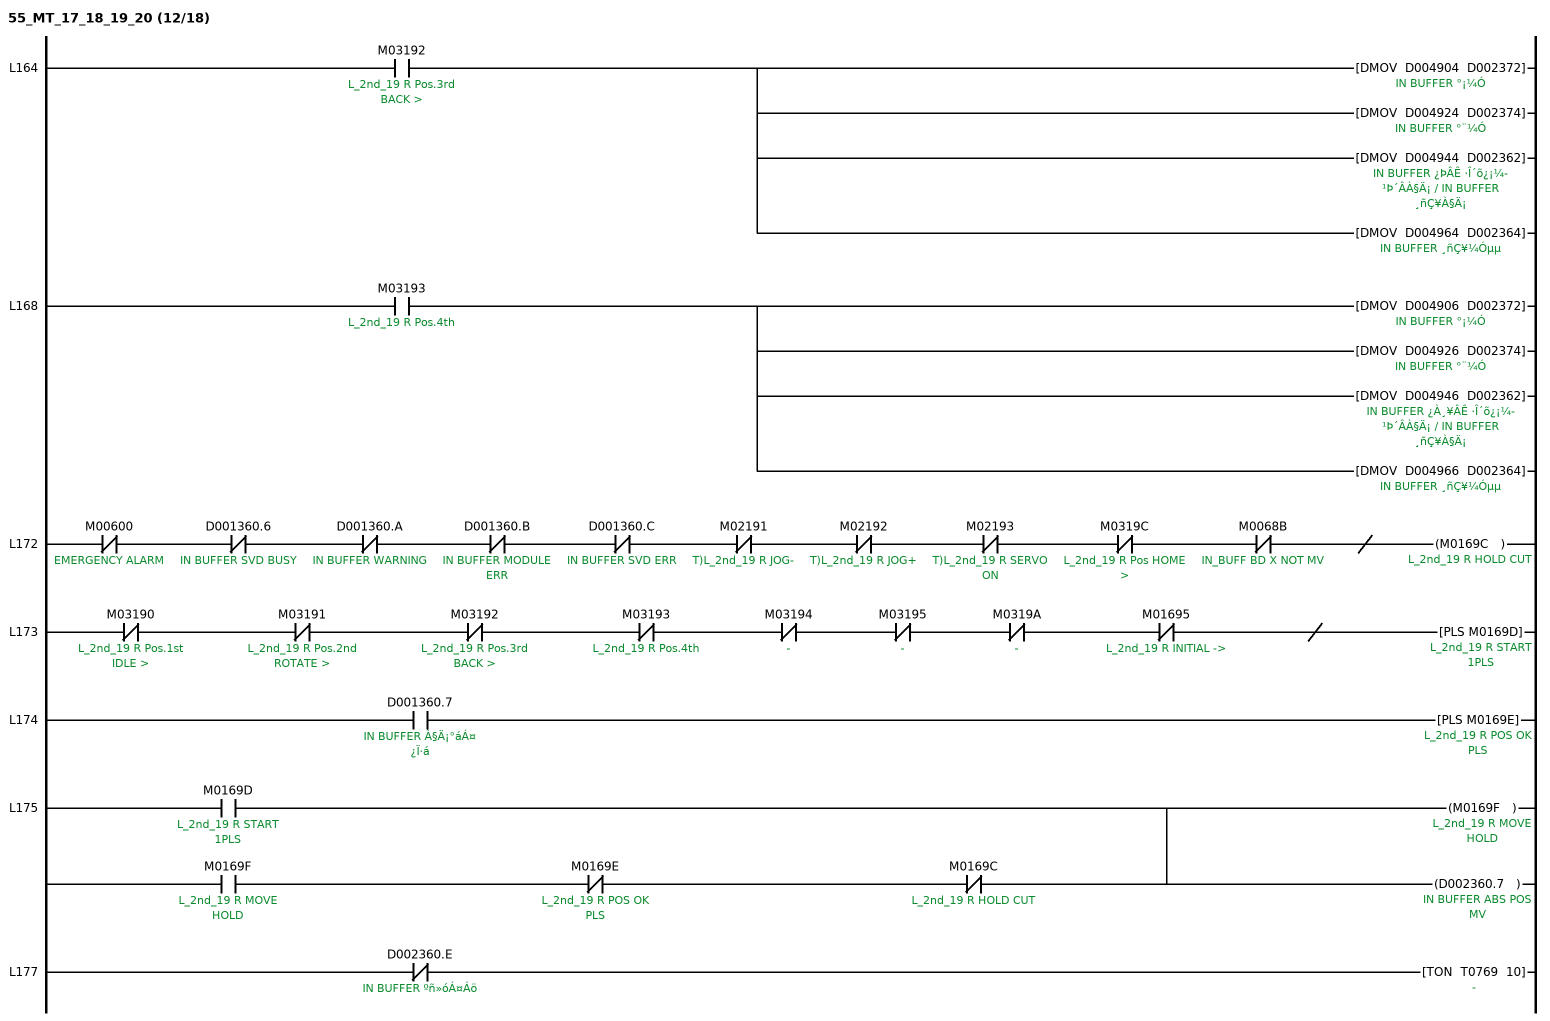
[picture p336: 55_MT_17_18_19_20 rungs L164-L177]
; L164
LOAD      M03192	// L_2nd_19 R Pos.3rd BACK >
DMOV      D004904 D002372	// IN BUFFER °¡¼Ó
DMOV      D004924 D002374	// IN BUFFER °¨¼Ó
DMOV      D004944 D002362	// IN BUFFER ¿ÞÂÊ ·Î´õ¿¡¼­ ¹Þ´ÂÀ§Ä¡ / IN BUFFER ¸ñÇ¥À§Ä¡
DMOV      D004964 D002364	// IN BUFFER ¸ñÇ¥¼Óµµ
; L168
LOAD      M03193	// L_2nd_19 R Pos.4th 
DMOV      D004906 D002372	// IN BUFFER °¡¼Ó
DMOV      D004926 D002374	// IN BUFFER °¨¼Ó
DMOV      D004946 D002362	// IN BUFFER ¿À¸¥ÂÊ ·Î´õ¿¡¼­ ¹Þ´ÂÀ§Ä¡ / IN BUFFER ¸ñÇ¥À§Ä¡
DMOV      D004966 D002364	// IN BUFFER ¸ñÇ¥¼Óµµ
; L172
LOAD NOT  M00600	// EMERGENCY ALARM
AND NOT   D001360.6	// IN BUFFER SVD BUSY
AND NOT   D001360.A	// IN BUFFER WARNING
AND NOT   D001360.B	// IN BUFFER MODULE ERR
AND NOT   D001360.C	// IN BUFFER SVD ERR
AND NOT   M02191	// T)L_2nd_19 R JOG-
AND NOT   M02192	// T)L_2nd_19 R JOG+
AND NOT   M02193	// T)L_2nd_19 R SERVO ON
AND NOT   M0319C	// L_2nd_19 R Pos HOME >
AND NOT   M0068B	// IN_BUFF BD X NOT MV
NOT
OUT       M0169C	// L_2nd_19 R HOLD CUT
; L173
LOAD NOT  M03190	// L_2nd_19 R Pos.1st IDLE >
AND NOT   M03191	// L_2nd_19 R Pos.2nd ROTATE >
AND NOT   M03192	// L_2nd_19 R Pos.3rd BACK >
AND NOT   M03193	// L_2nd_19 R Pos.4th 
AND NOT   M03194	// -
AND NOT   M03195	// -
AND NOT   M0319A	// -
AND NOT   M01695	// L_2nd_19 R INITIAL ->
NOT
OUTP      M0169D	// L_2nd_19 R START 1PLS
; L174
LOAD      D001360.7	// IN BUFFER À§Ä¡°áÁ¤ ¿Ï·á
OUTP      M0169E	// L_2nd_19 R POS OK PLS
; L175
LOAD      M0169D	// L_2nd_19 R START 1PLS
LOAD      M0169F	// L_2nd_19 R MOVE HOLD
AND NOT   M0169E	// L_2nd_19 R POS OK PLS
AND NOT   M0169C	// L_2nd_19 R HOLD CUT
OR LOAD
OUT       M0169F	// L_2nd_19 R MOVE HOLD
OUT       D002360.7	// IN BUFFER ABS POS MV
; L177
LOAD NOT  D002360.E	// IN BUFFER ºñ»óÁ¤Áö
TON       T0769 10	// -

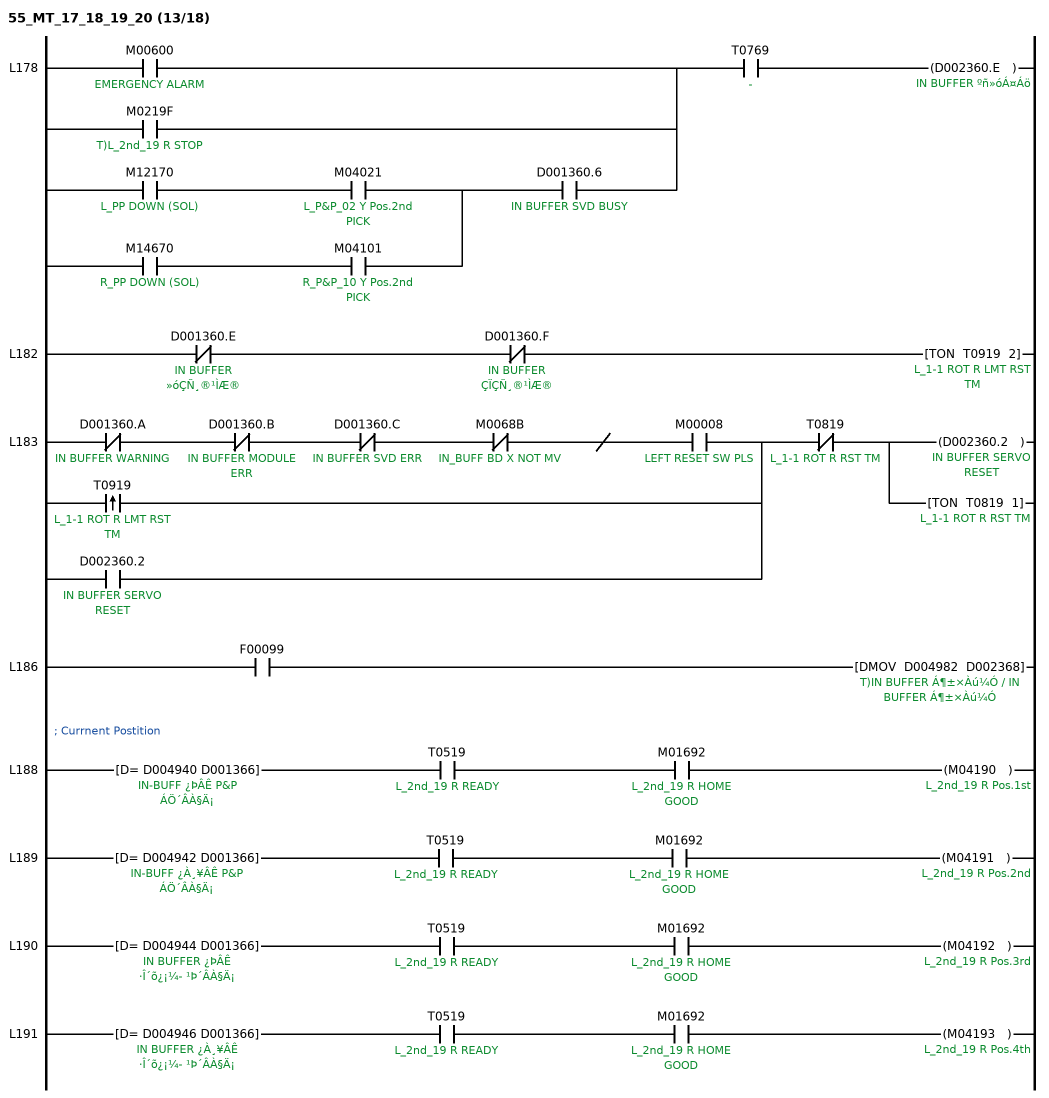
; L178
LOAD      M00600	// EMERGENCY ALARM
OR        M0219F	// T)L_2nd_19 R STOP
LOAD      M12170	// L_PP DOWN (SOL)
AND       M04021	// L_P&P_02 Y Pos.2nd PICK
LOAD      M14670	// R_PP DOWN (SOL)
AND       M04101	// R_P&P_10 Y Pos.2nd PICK
OR LOAD
AND       D001360.6	// IN BUFFER SVD BUSY
OR LOAD
AND       T0769	// -
OUT       D002360.E	// IN BUFFER ºñ»óÁ¤Áö
; L182
LOAD NOT  D001360.E	// IN BUFFER »óÇÑ¸®¹ÌÆ®
AND NOT   D001360.F	// IN BUFFER ÇÏÇÑ¸®¹ÌÆ®
TON       T0919 2	// L_1-1 ROT R LMT RST TM
; L183
LOAD NOT  D001360.A	// IN BUFFER WARNING
AND NOT   D001360.B	// IN BUFFER MODULE ERR
AND NOT   D001360.C	// IN BUFFER SVD ERR
AND NOT   M0068B	// IN_BUFF BD X NOT MV
NOT
AND       M00008	// LEFT RESET SW PLS
ORP       T0919	// L_1-1 ROT R LMT RST TM
OR        D002360.2	// IN BUFFER SERVO RESET
AND NOT   T0819	// L_1-1 ROT R RST TM
OUT       D002360.2	// IN BUFFER SERVO RESET
TON       T0819 1	// L_1-1 ROT R RST TM
; L186
LOAD      F00099
DMOV      D004982 D002368	// T)IN BUFFER Á¶±×Àú¼Ó / IN BUFFER Á¶±×Àú¼Ó
// Currnent Postition
; L188
LOADD=    D004940 D001366	// IN-BUFF ¿ÞÂÊ P&P ÁÖ´ÂÀ§Ä¡
AND       T0519	// L_2nd_19 R READY
AND       M01692	// L_2nd_19 R HOME GOOD
OUT       M04190	// L_2nd_19 R Pos.1st 
; L189
LOADD=    D004942 D001366	// IN-BUFF ¿À¸¥ÂÊ P&P ÁÖ´ÂÀ§Ä¡
AND       T0519	// L_2nd_19 R READY
AND       M01692	// L_2nd_19 R HOME GOOD
OUT       M04191	// L_2nd_19 R Pos.2nd
; L190
LOADD=    D004944 D001366	// IN BUFFER ¿ÞÂÊ ·Î´õ¿¡¼­ ¹Þ´ÂÀ§Ä¡
AND       T0519	// L_2nd_19 R READY
AND       M01692	// L_2nd_19 R HOME GOOD
OUT       M04192	// L_2nd_19 R Pos.3rd
; L191
LOADD=    D004946 D001366	// IN BUFFER ¿À¸¥ÂÊ ·Î´õ¿¡¼­ ¹Þ´ÂÀ§Ä¡
AND       T0519	// L_2nd_19 R READY
AND       M01692	// L_2nd_19 R HOME GOOD
OUT       M04193	// L_2nd_19 R Pos.4th 

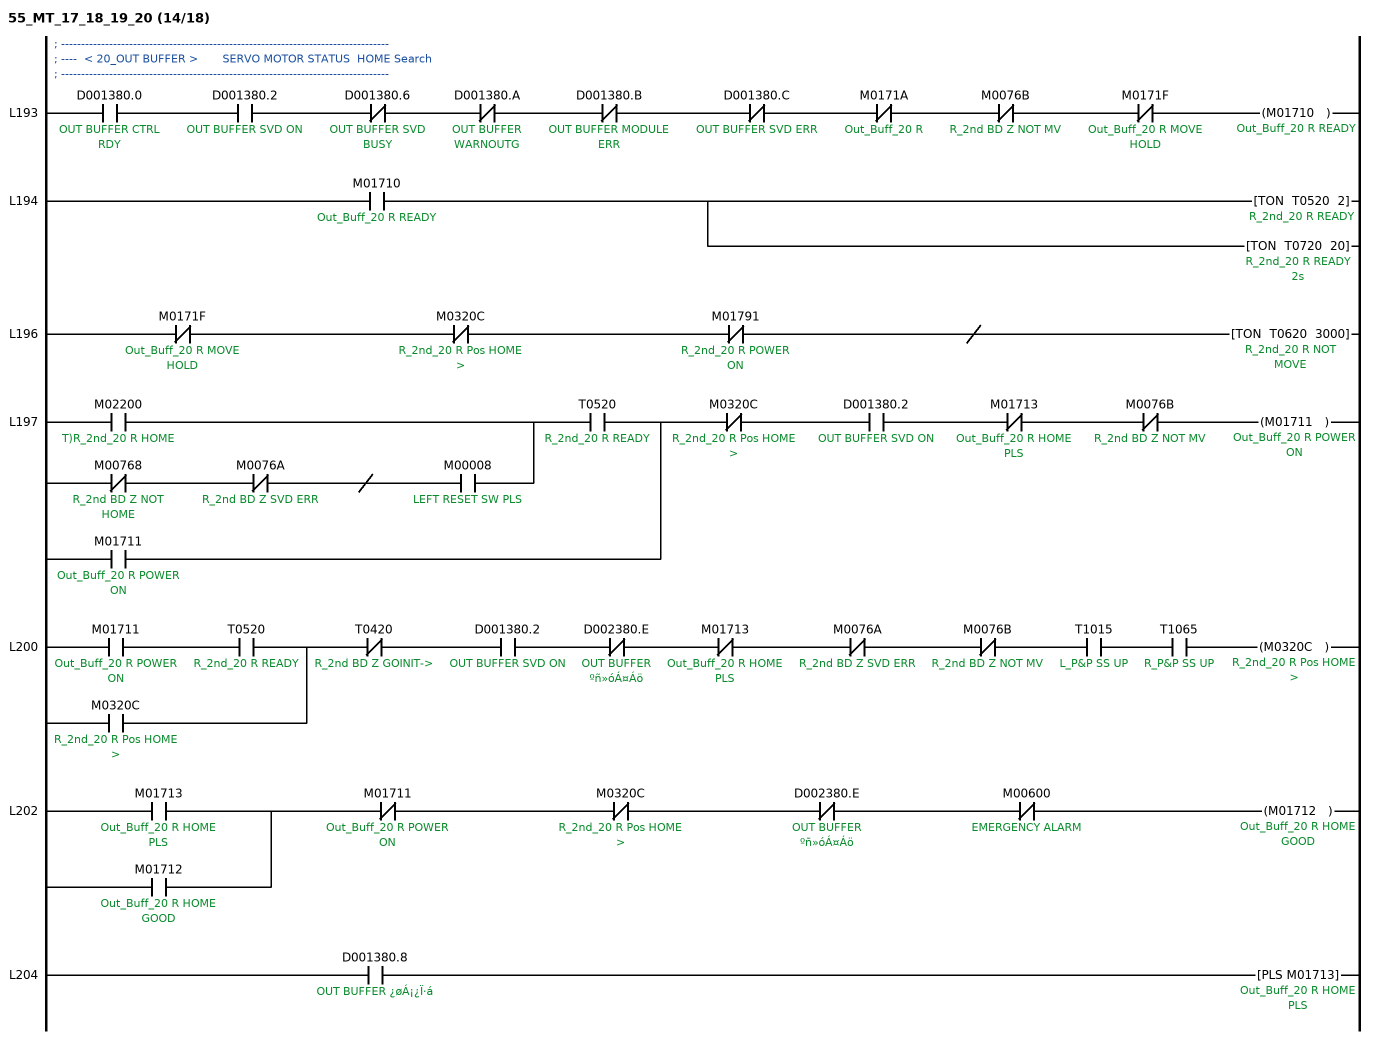
// ----------------------------------------------------------------------------------
// 
// ----  < 20_OUT BUFFER >       SERVO MOTOR STATUS  HOME Search
// 
// ----------------------------------------------------------------------------------
; L193
LOAD      D001380.0	// OUT BUFFER CTRL RDY
AND       D001380.2	// OUT BUFFER SVD ON
AND NOT   D001380.6	// OUT BUFFER SVD BUSY
AND NOT   D001380.A	// OUT BUFFER WARNOUTG
AND NOT   D001380.B	// OUT BUFFER MODULE ERR
AND NOT   D001380.C	// OUT BUFFER SVD ERR
AND NOT   M0171A	// Out_Buff_20 R
AND NOT   M0076B	// R_2nd BD Z NOT MV
AND NOT   M0171F	// Out_Buff_20 R MOVE HOLD
OUT       M01710	// Out_Buff_20 R READY
; L194
LOAD      M01710	// Out_Buff_20 R READY
TON       T0520 2	// R_2nd_20 R READY
TON       T0720 20	// R_2nd_20 R READY 2s
; L196
LOAD NOT  M0171F	// Out_Buff_20 R MOVE HOLD
AND NOT   M0320C	// R_2nd_20 R Pos HOME >
AND NOT   M01791	// R_2nd_20 R POWER ON
NOT
TON       T0620 3000	// R_2nd_20 R NOT MOVE
; L197
LOAD      M02200	// T)R_2nd_20 R HOME
LOAD NOT  M00768	// R_2nd BD Z NOT HOME
AND NOT   M0076A	// R_2nd BD Z SVD ERR
NOT
AND       M00008	// LEFT RESET SW PLS
OR LOAD
AND       T0520	// R_2nd_20 R READY
OR        M01711	// Out_Buff_20 R POWER ON
AND NOT   M0320C	// R_2nd_20 R Pos HOME >
AND       D001380.2	// OUT BUFFER SVD ON
AND NOT   M01713	// Out_Buff_20 R HOME PLS
AND NOT   M0076B	// R_2nd BD Z NOT MV
OUT       M01711	// Out_Buff_20 R POWER ON
; L200
LOAD      M01711	// Out_Buff_20 R POWER ON
AND       T0520	// R_2nd_20 R READY
OR        M0320C	// R_2nd_20 R Pos HOME >
AND NOT   T0420	// R_2nd BD Z GOINIT->
AND       D001380.2	// OUT BUFFER SVD ON
AND NOT   D002380.E	// OUT BUFFER ºñ»óÁ¤Áö
AND NOT   M01713	// Out_Buff_20 R HOME PLS
AND NOT   M0076A	// R_2nd BD Z SVD ERR
AND NOT   M0076B	// R_2nd BD Z NOT MV
AND       T1015	// L_P&P SS UP
AND       T1065	// R_P&P SS UP
OUT       M0320C	// R_2nd_20 R Pos HOME >
; L202
LOAD      M01713	// Out_Buff_20 R HOME PLS
OR        M01712	// Out_Buff_20 R HOME GOOD
AND NOT   M01711	// Out_Buff_20 R POWER ON
AND NOT   M0320C	// R_2nd_20 R Pos HOME >
AND NOT   D002380.E	// OUT BUFFER ºñ»óÁ¤Áö
AND NOT   M00600	// EMERGENCY ALARM
OUT       M01712	// Out_Buff_20 R HOME GOOD
; L204
LOAD      D001380.8	// OUT BUFFER ¿øÁ¡¿Ï·á
OUTP      M01713	// Out_Buff_20 R HOME PLS

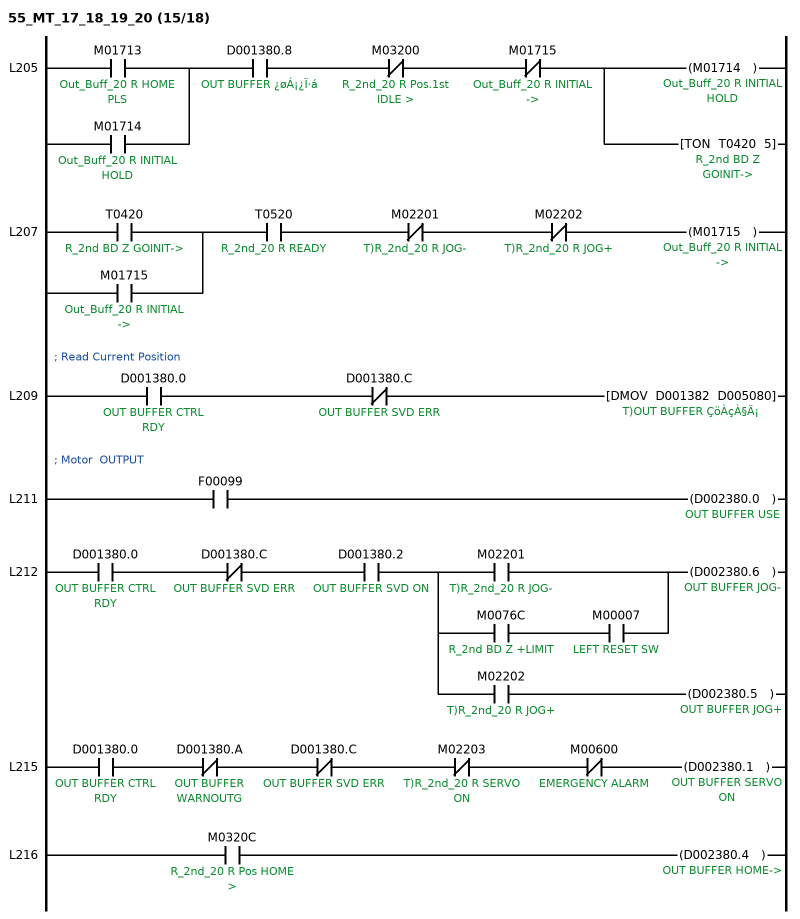
; L205
LOAD      M01713	// Out_Buff_20 R HOME PLS
OR        M01714	// Out_Buff_20 R INITIAL HOLD
AND       D001380.8	// OUT BUFFER ¿øÁ¡¿Ï·á
AND NOT   M03200	// R_2nd_20 R Pos.1st IDLE >
AND NOT   M01715	// Out_Buff_20 R INITIAL ->
OUT       M01714	// Out_Buff_20 R INITIAL HOLD
TON       T0420 5	// R_2nd BD Z GOINIT->
; L207
LOAD      T0420	// R_2nd BD Z GOINIT->
OR        M01715	// Out_Buff_20 R INITIAL ->
AND       T0520	// R_2nd_20 R READY
AND NOT   M02201	// T)R_2nd_20 R JOG-
AND NOT   M02202	// T)R_2nd_20 R JOG+
OUT       M01715	// Out_Buff_20 R INITIAL ->
; L209
LOAD      D001380.0	// OUT BUFFER CTRL RDY
AND NOT   D001380.C	// OUT BUFFER SVD ERR
DMOV      D001382 D005080	// T)OUT BUFFER ÇöÀçÀ§Ä¡
// output comment: Read Current Position
//  Motor  OUTPUT
; L211
LOAD      F00099
OUT       D002380.0	// OUT BUFFER USE
; L212
LOAD      D001380.0	// OUT BUFFER CTRL RDY
AND NOT   D001380.C	// OUT BUFFER SVD ERR
AND       D001380.2	// OUT BUFFER SVD ON
MPUSH
LOAD      M02201	// T)R_2nd_20 R JOG-
LOAD      M0076C	// R_2nd BD Z +LIMIT
AND       M00007	// LEFT RESET SW
OR LOAD
AND LOAD
OUT       D002380.6	// OUT BUFFER JOG-
MPOP
AND       M02202	// T)R_2nd_20 R JOG+
OUT       D002380.5	// OUT BUFFER JOG+
; L215
LOAD      D001380.0	// OUT BUFFER CTRL RDY
AND NOT   D001380.A	// OUT BUFFER WARNOUTG
AND NOT   D001380.C	// OUT BUFFER SVD ERR
AND NOT   M02203	// T)R_2nd_20 R SERVO ON
AND NOT   M00600	// EMERGENCY ALARM
OUT       D002380.1	// OUT BUFFER SERVO ON
; L216
LOAD      M0320C	// R_2nd_20 R Pos HOME >
OUT       D002380.4	// OUT BUFFER HOME->

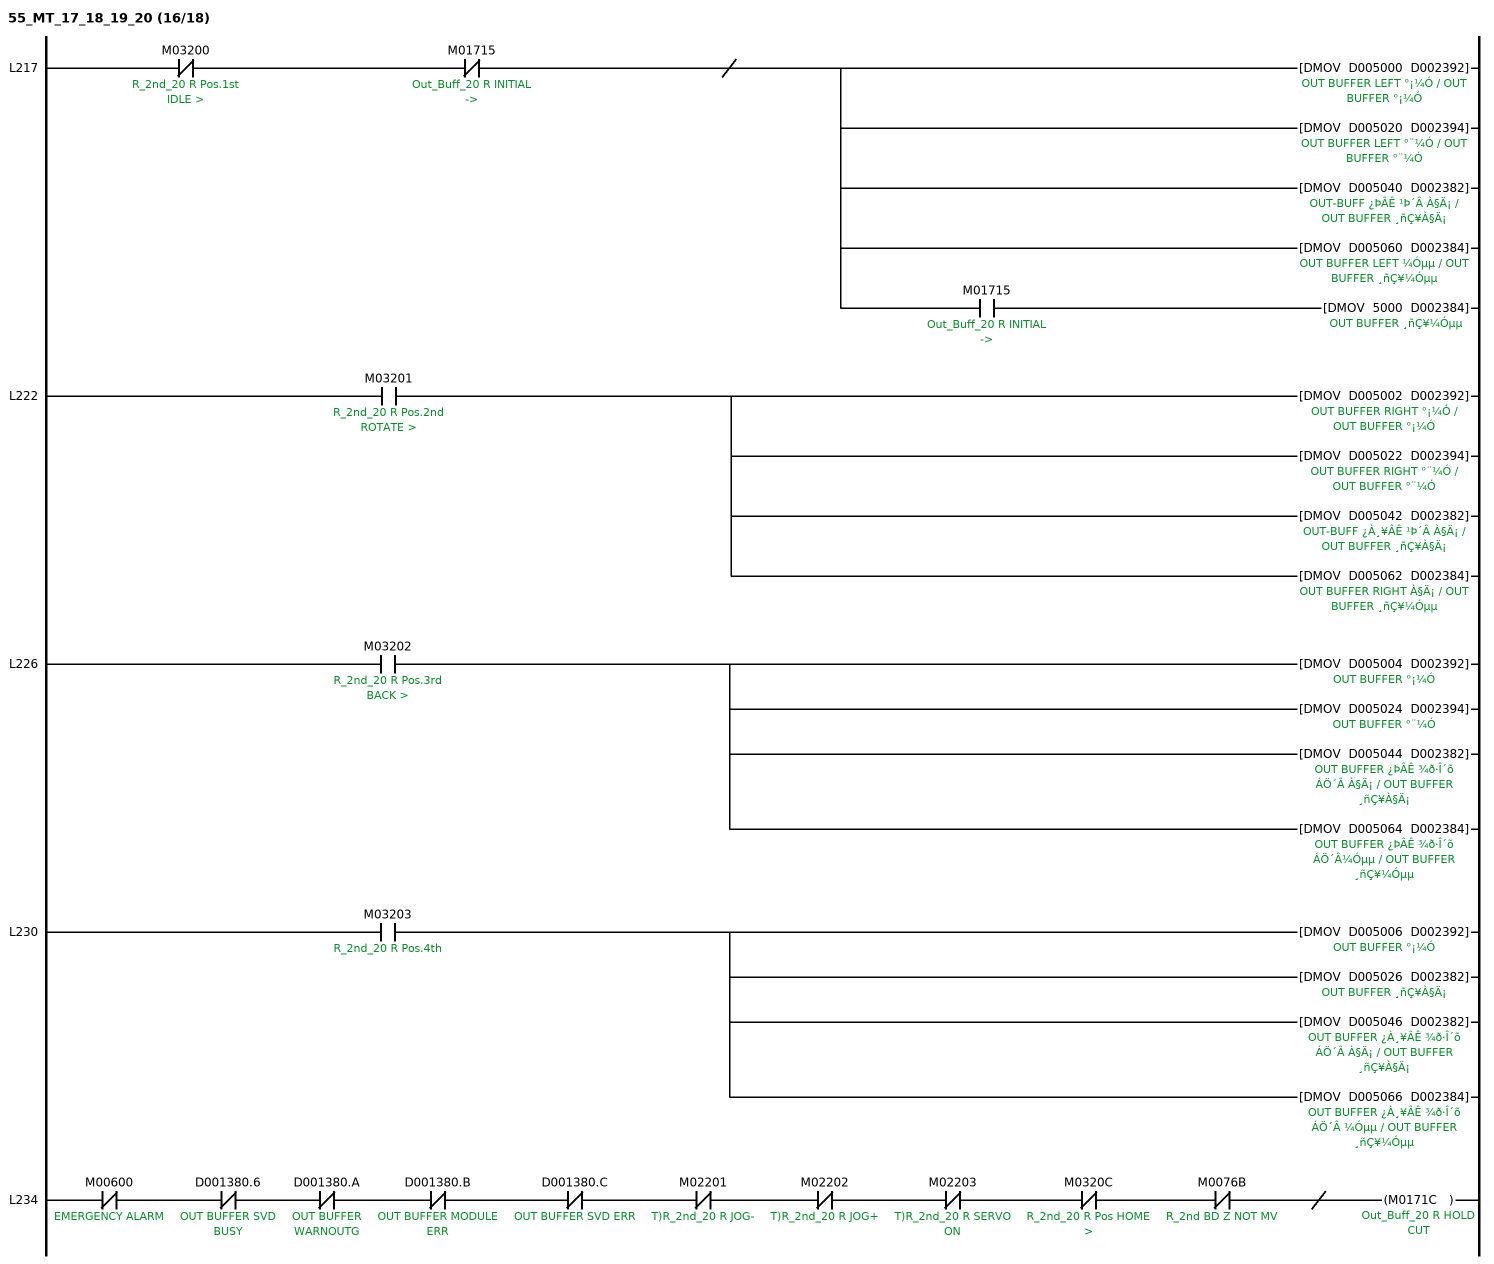
; L217
LOAD NOT  M03200	// R_2nd_20 R Pos.1st IDLE >
AND NOT   M01715	// Out_Buff_20 R INITIAL ->
NOT
DMOV      D005000 D002392	// OUT BUFFER LEFT °¡¼Ó / OUT BUFFER °¡¼Ó
DMOV      D005020 D002394	// OUT BUFFER LEFT °¨¼Ó / OUT BUFFER °¨¼Ó
DMOV      D005040 D002382	// OUT-BUFF ¿ÞÂÊ ¹Þ´Â À§Ä¡ / OUT BUFFER ¸ñÇ¥À§Ä¡
DMOV      D005060 D002384	// OUT BUFFER LEFT ¼Óµµ / OUT BUFFER ¸ñÇ¥¼Óµµ
AND       M01715	// Out_Buff_20 R INITIAL ->
DMOV      5000 D002384	// OUT BUFFER ¸ñÇ¥¼Óµµ
; L222
LOAD      M03201	// R_2nd_20 R Pos.2nd ROTATE >
DMOV      D005002 D002392	// OUT BUFFER RIGHT °¡¼Ó / OUT BUFFER °¡¼Ó
DMOV      D005022 D002394	// OUT BUFFER RIGHT °¨¼Ó / OUT BUFFER °¨¼Ó
DMOV      D005042 D002382	// OUT-BUFF ¿À¸¥ÂÊ ¹Þ´Â À§Ä¡ / OUT BUFFER ¸ñÇ¥À§Ä¡
DMOV      D005062 D002384	// OUT BUFFER RIGHT À§Ä¡ / OUT BUFFER ¸ñÇ¥¼Óµµ
; L226
LOAD      M03202	// R_2nd_20 R Pos.3rd BACK >
DMOV      D005004 D002392	// OUT BUFFER °¡¼Ó
DMOV      D005024 D002394	// OUT BUFFER °¨¼Ó
DMOV      D005044 D002382	// OUT BUFFER ¿ÞÂÊ ¾ð·Î´õ ÁÖ´Â À§Ä¡ / OUT BUFFER ¸ñÇ¥À§Ä¡
DMOV      D005064 D002384	// OUT BUFFER ¿ÞÂÊ ¾ð·Î´õ ÁÖ´Â¼Óµµ / OUT BUFFER ¸ñÇ¥¼Óµµ
; L230
LOAD      M03203	// R_2nd_20 R Pos.4th 
DMOV      D005006 D002392	// OUT BUFFER °¡¼Ó
DMOV      D005026 D002382	// OUT BUFFER ¸ñÇ¥À§Ä¡
DMOV      D005046 D002382	// OUT BUFFER ¿À¸¥ÂÊ ¾ð·Î´õ ÁÖ´Â À§Ä¡ / OUT BUFFER ¸ñÇ¥À§Ä¡
DMOV      D005066 D002384	// OUT BUFFER ¿À¸¥ÂÊ ¾ð·Î´õ ÁÖ´Â ¼Óµµ / OUT BUFFER ¸ñÇ¥¼Óµµ
; L234
LOAD NOT  M00600	// EMERGENCY ALARM
AND NOT   D001380.6	// OUT BUFFER SVD BUSY
AND NOT   D001380.A	// OUT BUFFER WARNOUTG
AND NOT   D001380.B	// OUT BUFFER MODULE ERR
AND NOT   D001380.C	// OUT BUFFER SVD ERR
AND NOT   M02201	// T)R_2nd_20 R JOG-
AND NOT   M02202	// T)R_2nd_20 R JOG+
AND NOT   M02203	// T)R_2nd_20 R SERVO ON
AND NOT   M0320C	// R_2nd_20 R Pos HOME >
AND NOT   M0076B	// R_2nd BD Z NOT MV
NOT
OUT       M0171C	// Out_Buff_20 R HOLD CUT

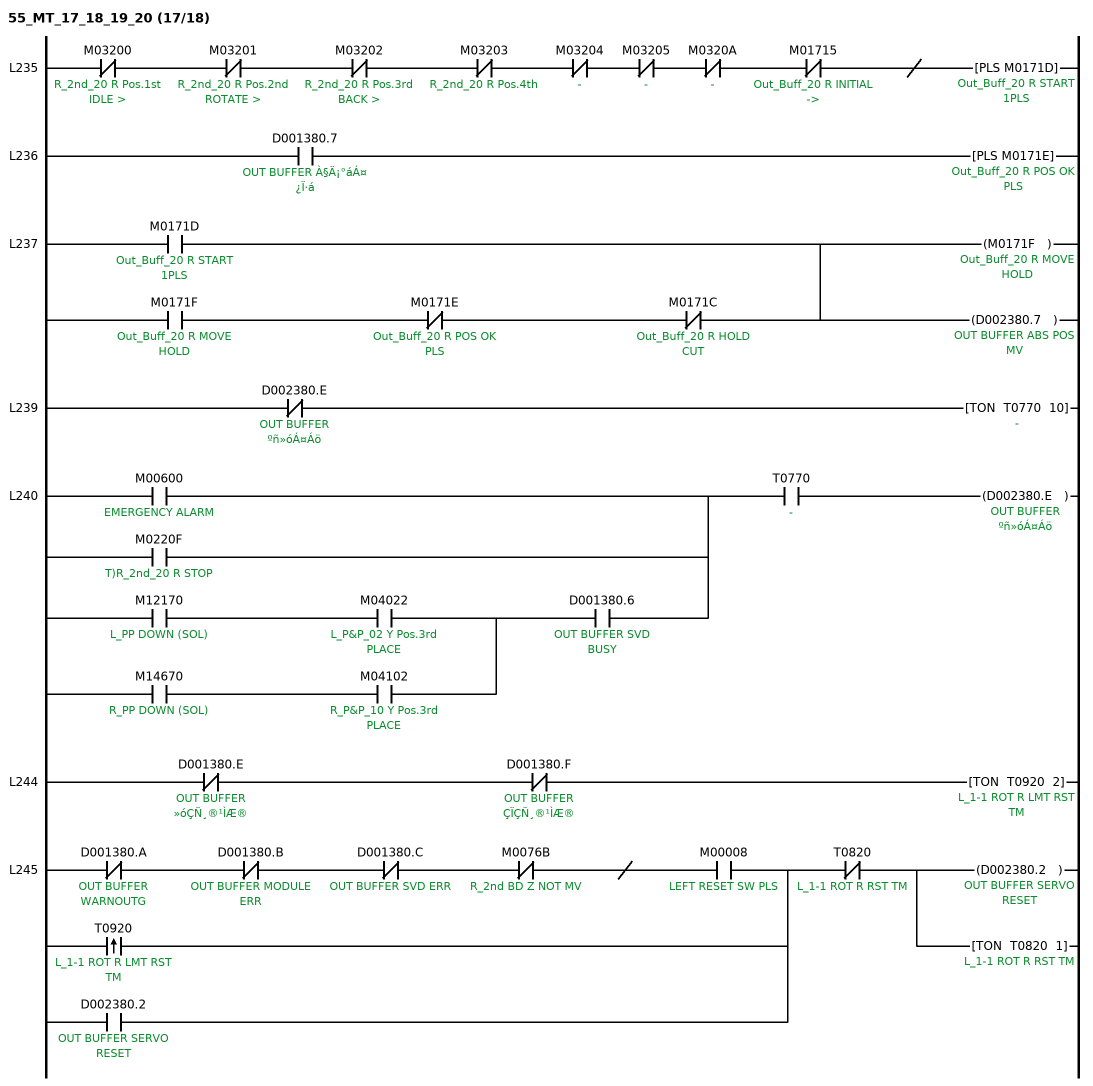
; L235
LOAD NOT  M03200	// R_2nd_20 R Pos.1st IDLE >
AND NOT   M03201	// R_2nd_20 R Pos.2nd ROTATE >
AND NOT   M03202	// R_2nd_20 R Pos.3rd BACK >
AND NOT   M03203	// R_2nd_20 R Pos.4th 
AND NOT   M03204	// -
AND NOT   M03205	// -
AND NOT   M0320A	// -
AND NOT   M01715	// Out_Buff_20 R INITIAL ->
NOT
OUTP      M0171D	// Out_Buff_20 R START 1PLS
; L236
LOAD      D001380.7	// OUT BUFFER À§Ä¡°áÁ¤ ¿Ï·á
OUTP      M0171E	// Out_Buff_20 R POS OK PLS
; L237
LOAD      M0171D	// Out_Buff_20 R START 1PLS
LOAD      M0171F	// Out_Buff_20 R MOVE HOLD
AND NOT   M0171E	// Out_Buff_20 R POS OK PLS
AND NOT   M0171C	// Out_Buff_20 R HOLD CUT
OR LOAD
OUT       M0171F	// Out_Buff_20 R MOVE HOLD
OUT       D002380.7	// OUT BUFFER ABS POS MV
; L239
LOAD NOT  D002380.E	// OUT BUFFER ºñ»óÁ¤Áö
TON       T0770 10	// -
; L240
LOAD      M00600	// EMERGENCY ALARM
OR        M0220F	// T)R_2nd_20 R STOP
LOAD      M12170	// L_PP DOWN (SOL)
AND       M04022	// L_P&P_02 Y Pos.3rd PLACE
LOAD      M14670	// R_PP DOWN (SOL)
AND       M04102	// R_P&P_10 Y Pos.3rd PLACE
OR LOAD
AND       D001380.6	// OUT BUFFER SVD BUSY
OR LOAD
AND       T0770	// -
OUT       D002380.E	// OUT BUFFER ºñ»óÁ¤Áö
; L244
LOAD NOT  D001380.E	// OUT BUFFER »óÇÑ¸®¹ÌÆ®
AND NOT   D001380.F	// OUT BUFFER ÇÏÇÑ¸®¹ÌÆ®
TON       T0920 2	// L_1-1 ROT R LMT RST TM
; L245
LOAD NOT  D001380.A	// OUT BUFFER WARNOUTG
AND NOT   D001380.B	// OUT BUFFER MODULE ERR
AND NOT   D001380.C	// OUT BUFFER SVD ERR
AND NOT   M0076B	// R_2nd BD Z NOT MV
NOT
AND       M00008	// LEFT RESET SW PLS
ORP       T0920	// L_1-1 ROT R LMT RST TM
OR        D002380.2	// OUT BUFFER SERVO RESET
AND NOT   T0820	// L_1-1 ROT R RST TM
OUT       D002380.2	// OUT BUFFER SERVO RESET
TON       T0820 1	// L_1-1 ROT R RST TM

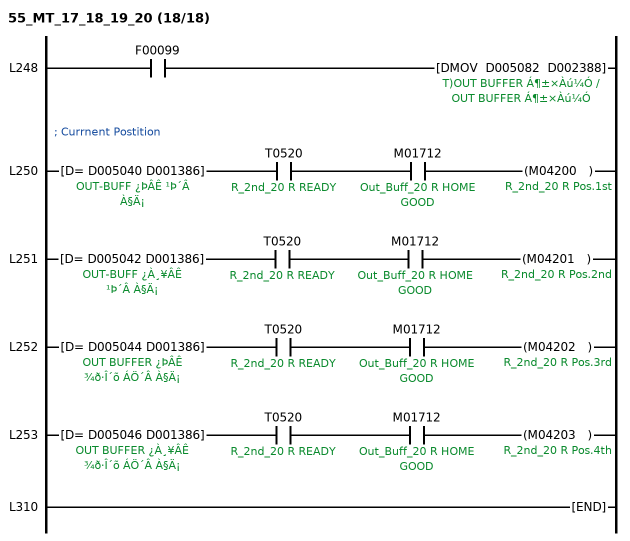
; L248
LOAD      F00099
DMOV      D005082 D002388	// T)OUT BUFFER Á¶±×Àú¼Ó / OUT BUFFER Á¶±×Àú¼Ó
// Currnent Postition
; L250
LOADD=    D005040 D001386	// OUT-BUFF ¿ÞÂÊ ¹Þ´Â À§Ä¡
AND       T0520	// R_2nd_20 R READY
AND       M01712	// Out_Buff_20 R HOME GOOD
OUT       M04200	// R_2nd_20 R Pos.1st
; L251
LOADD=    D005042 D001386	// OUT-BUFF ¿À¸¥ÂÊ ¹Þ´Â À§Ä¡
AND       T0520	// R_2nd_20 R READY
AND       M01712	// Out_Buff_20 R HOME GOOD
OUT       M04201	// R_2nd_20 R Pos.2nd
; L252
LOADD=    D005044 D001386	// OUT BUFFER ¿ÞÂÊ ¾ð·Î´õ ÁÖ´Â À§Ä¡
AND       T0520	// R_2nd_20 R READY
AND       M01712	// Out_Buff_20 R HOME GOOD
OUT       M04202	// R_2nd_20 R Pos.3rd
; L253
LOADD=    D005046 D001386	// OUT BUFFER ¿À¸¥ÂÊ ¾ð·Î´õ ÁÖ´Â À§Ä¡
AND       T0520	// R_2nd_20 R READY
AND       M01712	// Out_Buff_20 R HOME GOOD
OUT       M04203	// R_2nd_20 R Pos.4th 
; L310
END

PROGRAM 56_MT_21_22_23_24 (task: ½ºÄµ ÇÁ·Î±×·¥)

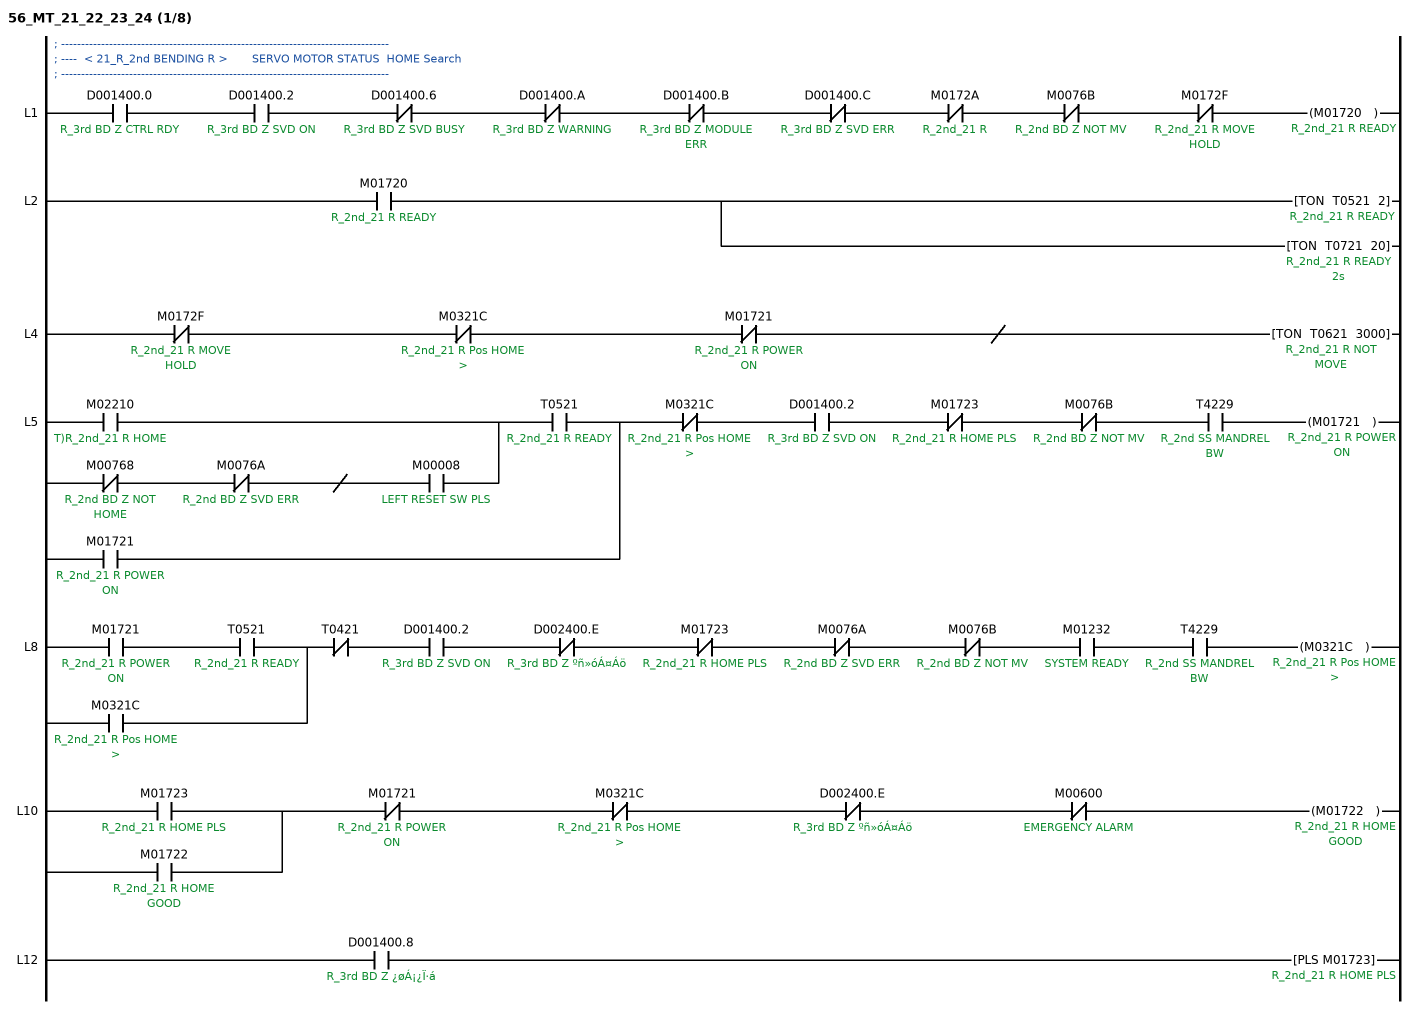
// ----------------------------------------------------------------------------------
// 
// ----  < 21_R_2nd BENDING R >       SERVO MOTOR STATUS  HOME Search
// 
// ----------------------------------------------------------------------------------
; L1
LOAD      D001400.0	// R_3rd BD Z CTRL RDY
AND       D001400.2	// R_3rd BD Z SVD ON
AND NOT   D001400.6	// R_3rd BD Z SVD BUSY
AND NOT   D001400.A	// R_3rd BD Z WARNING
AND NOT   D001400.B	// R_3rd BD Z MODULE ERR
AND NOT   D001400.C	// R_3rd BD Z SVD ERR
AND NOT   M0172A	// R_2nd_21 R
AND NOT   M0076B	// R_2nd BD Z NOT MV
AND NOT   M0172F	// R_2nd_21 R MOVE HOLD
OUT       M01720	// R_2nd_21 R READY
; L2
LOAD      M01720	// R_2nd_21 R READY
TON       T0521 2	// R_2nd_21 R READY
TON       T0721 20	// R_2nd_21 R READY 2s
; L4
LOAD NOT  M0172F	// R_2nd_21 R MOVE HOLD
AND NOT   M0321C	// R_2nd_21 R Pos HOME >
AND NOT   M01721	// R_2nd_21 R POWER ON
NOT
TON       T0621 3000	// R_2nd_21 R NOT MOVE
; L5
LOAD      M02210	// T)R_2nd_21 R HOME
LOAD NOT  M00768	// R_2nd BD Z NOT HOME
AND NOT   M0076A	// R_2nd BD Z SVD ERR
NOT
AND       M00008	// LEFT RESET SW PLS
OR LOAD
AND       T0521	// R_2nd_21 R READY
OR        M01721	// R_2nd_21 R POWER ON
AND NOT   M0321C	// R_2nd_21 R Pos HOME >
AND       D001400.2	// R_3rd BD Z SVD ON
AND NOT   M01723	// R_2nd_21 R HOME PLS
AND NOT   M0076B	// R_2nd BD Z NOT MV
AND       T4229	// R_2nd SS MANDREL BW
OUT       M01721	// R_2nd_21 R POWER ON
; L8
LOAD      M01721	// R_2nd_21 R POWER ON
AND       T0521	// R_2nd_21 R READY
OR        M0321C	// R_2nd_21 R Pos HOME >
AND NOT   T0421
AND       D001400.2	// R_3rd BD Z SVD ON
AND NOT   D002400.E	// R_3rd BD Z ºñ»óÁ¤Áö
AND NOT   M01723	// R_2nd_21 R HOME PLS
AND NOT   M0076A	// R_2nd BD Z SVD ERR
AND NOT   M0076B	// R_2nd BD Z NOT MV
AND       M01232	// SYSTEM READY
AND       T4229	// R_2nd SS MANDREL BW
OUT       M0321C	// R_2nd_21 R Pos HOME >
; L10
LOAD      M01723	// R_2nd_21 R HOME PLS
OR        M01722	// R_2nd_21 R HOME GOOD
AND NOT   M01721	// R_2nd_21 R POWER ON
AND NOT   M0321C	// R_2nd_21 R Pos HOME >
AND NOT   D002400.E	// R_3rd BD Z ºñ»óÁ¤Áö
AND NOT   M00600	// EMERGENCY ALARM
OUT       M01722	// R_2nd_21 R HOME GOOD
; L12
LOAD      D001400.8	// R_3rd BD Z ¿øÁ¡¿Ï·á
OUTP      M01723	// R_2nd_21 R HOME PLS

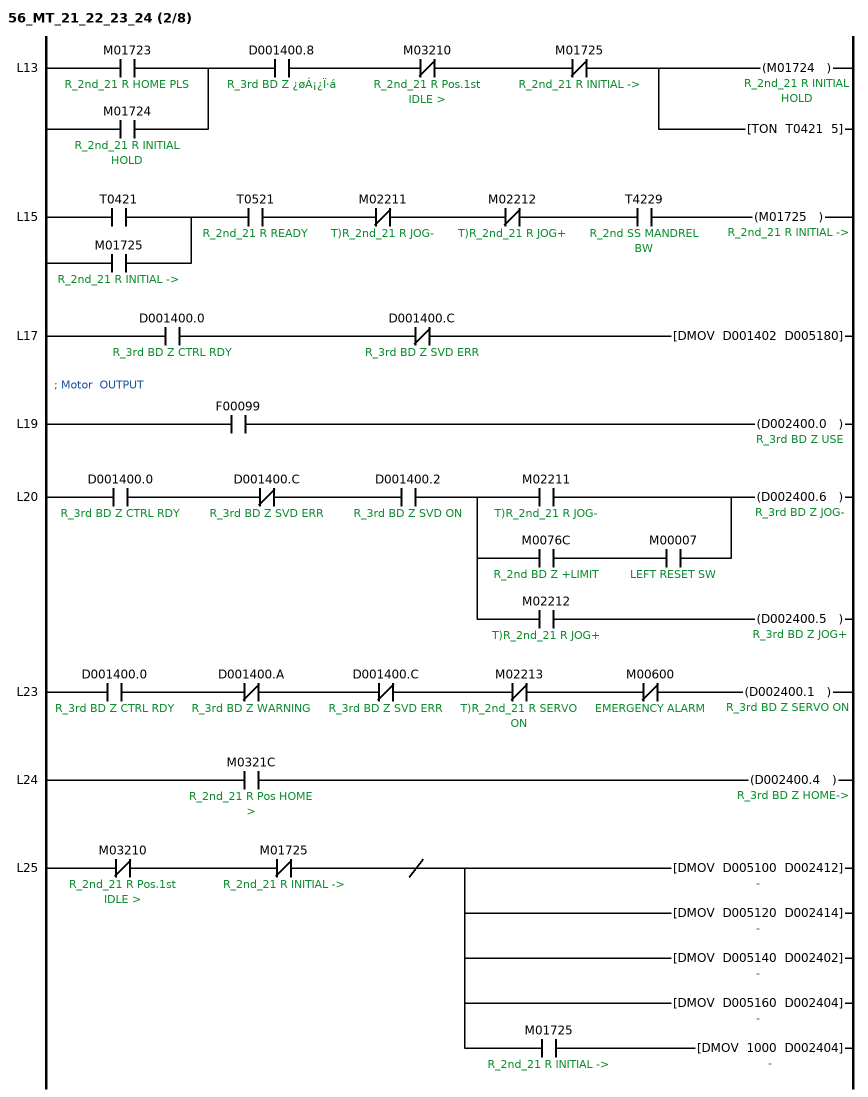
; L13
LOAD      M01723	// R_2nd_21 R HOME PLS
OR        M01724	// R_2nd_21 R INITIAL HOLD
AND       D001400.8	// R_3rd BD Z ¿øÁ¡¿Ï·á
AND NOT   M03210	// R_2nd_21 R Pos.1st IDLE >
AND NOT   M01725	// R_2nd_21 R INITIAL ->
OUT       M01724	// R_2nd_21 R INITIAL HOLD
TON       T0421 5
; L15
LOAD      T0421
OR        M01725	// R_2nd_21 R INITIAL ->
AND       T0521	// R_2nd_21 R READY
AND NOT   M02211	// T)R_2nd_21 R JOG-
AND NOT   M02212	// T)R_2nd_21 R JOG+
AND       T4229	// R_2nd SS MANDREL BW
OUT       M01725	// R_2nd_21 R INITIAL ->
; L17
LOAD      D001400.0	// R_3rd BD Z CTRL RDY
AND NOT   D001400.C	// R_3rd BD Z SVD ERR
DMOV      D001402 D005180
//  Motor  OUTPUT
; L19
LOAD      F00099
OUT       D002400.0	// R_3rd BD Z USE
; L20
LOAD      D001400.0	// R_3rd BD Z CTRL RDY
AND NOT   D001400.C	// R_3rd BD Z SVD ERR
AND       D001400.2	// R_3rd BD Z SVD ON
MPUSH
LOAD      M02211	// T)R_2nd_21 R JOG-
LOAD      M0076C	// R_2nd BD Z +LIMIT
AND       M00007	// LEFT RESET SW
OR LOAD
AND LOAD
OUT       D002400.6	// R_3rd BD Z JOG-
MPOP
AND       M02212	// T)R_2nd_21 R JOG+
OUT       D002400.5	// R_3rd BD Z JOG+
; L23
LOAD      D001400.0	// R_3rd BD Z CTRL RDY
AND NOT   D001400.A	// R_3rd BD Z WARNING
AND NOT   D001400.C	// R_3rd BD Z SVD ERR
AND NOT   M02213	// T)R_2nd_21 R SERVO ON
AND NOT   M00600	// EMERGENCY ALARM
OUT       D002400.1	// R_3rd BD Z SERVO ON
; L24
LOAD      M0321C	// R_2nd_21 R Pos HOME >
OUT       D002400.4	// R_3rd BD Z HOME->
; L25
LOAD NOT  M03210	// R_2nd_21 R Pos.1st IDLE >
AND NOT   M01725	// R_2nd_21 R INITIAL ->
NOT
DMOV      D005100 D002412	// -
DMOV      D005120 D002414	// -
DMOV      D005140 D002402	// -
DMOV      D005160 D002404	// -
AND       M01725	// R_2nd_21 R INITIAL ->
DMOV      1000 D002404	// -

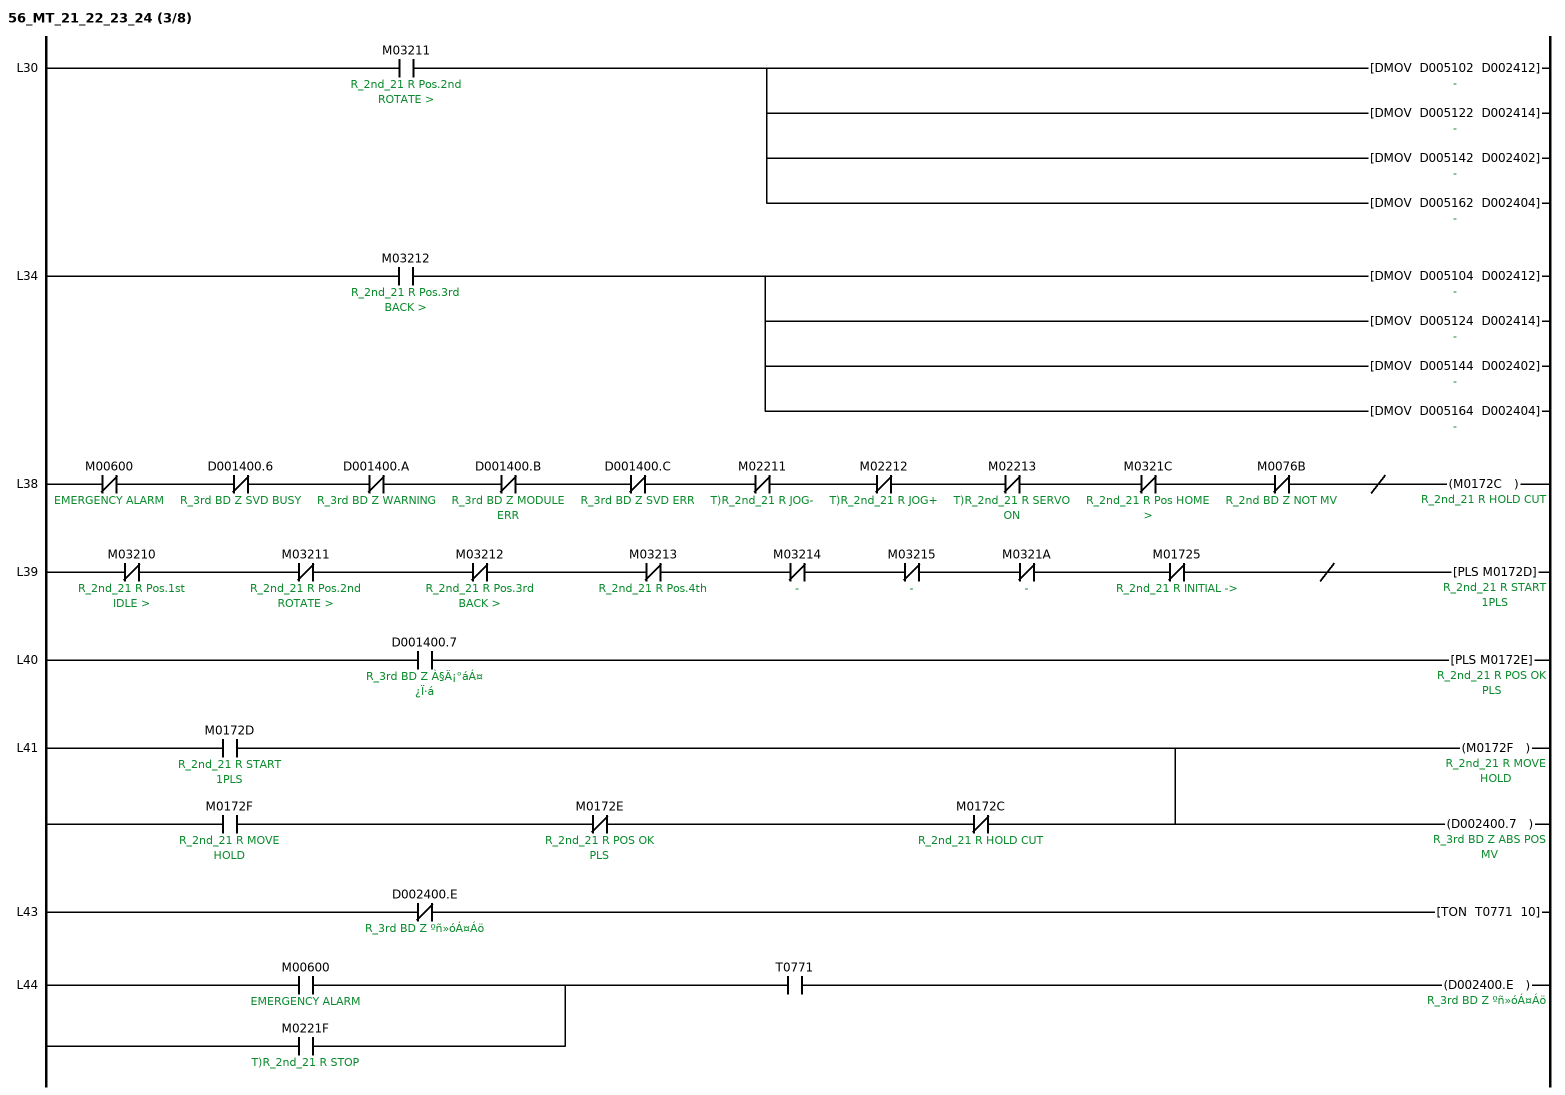
; L30
LOAD      M03211	// R_2nd_21 R Pos.2nd ROTATE >
DMOV      D005102 D002412	// -
DMOV      D005122 D002414	// -
DMOV      D005142 D002402	// -
DMOV      D005162 D002404	// -
; L34
LOAD      M03212	// R_2nd_21 R Pos.3rd BACK >
DMOV      D005104 D002412	// -
DMOV      D005124 D002414	// -
DMOV      D005144 D002402	// -
DMOV      D005164 D002404	// -
; L38
LOAD NOT  M00600	// EMERGENCY ALARM
AND NOT   D001400.6	// R_3rd BD Z SVD BUSY
AND NOT   D001400.A	// R_3rd BD Z WARNING
AND NOT   D001400.B	// R_3rd BD Z MODULE ERR
AND NOT   D001400.C	// R_3rd BD Z SVD ERR
AND NOT   M02211	// T)R_2nd_21 R JOG-
AND NOT   M02212	// T)R_2nd_21 R JOG+
AND NOT   M02213	// T)R_2nd_21 R SERVO ON
AND NOT   M0321C	// R_2nd_21 R Pos HOME >
AND NOT   M0076B	// R_2nd BD Z NOT MV
NOT
OUT       M0172C	// R_2nd_21 R HOLD CUT
; L39
LOAD NOT  M03210	// R_2nd_21 R Pos.1st IDLE >
AND NOT   M03211	// R_2nd_21 R Pos.2nd ROTATE >
AND NOT   M03212	// R_2nd_21 R Pos.3rd BACK >
AND NOT   M03213	// R_2nd_21 R Pos.4th 
AND NOT   M03214	// -
AND NOT   M03215	// -
AND NOT   M0321A	// -
AND NOT   M01725	// R_2nd_21 R INITIAL ->
NOT
OUTP      M0172D	// R_2nd_21 R START 1PLS
; L40
LOAD      D001400.7	// R_3rd BD Z À§Ä¡°áÁ¤ ¿Ï·á
OUTP      M0172E	// R_2nd_21 R POS OK PLS
; L41
LOAD      M0172D	// R_2nd_21 R START 1PLS
LOAD      M0172F	// R_2nd_21 R MOVE HOLD
AND NOT   M0172E	// R_2nd_21 R POS OK PLS
AND NOT   M0172C	// R_2nd_21 R HOLD CUT
OR LOAD
OUT       M0172F	// R_2nd_21 R MOVE HOLD
OUT       D002400.7	// R_3rd BD Z ABS POS MV
; L43
LOAD NOT  D002400.E	// R_3rd BD Z ºñ»óÁ¤Áö
TON       T0771 10
; L44
LOAD      M00600	// EMERGENCY ALARM
OR        M0221F	// T)R_2nd_21 R STOP
AND       T0771
OUT       D002400.E	// R_3rd BD Z ºñ»óÁ¤Áö

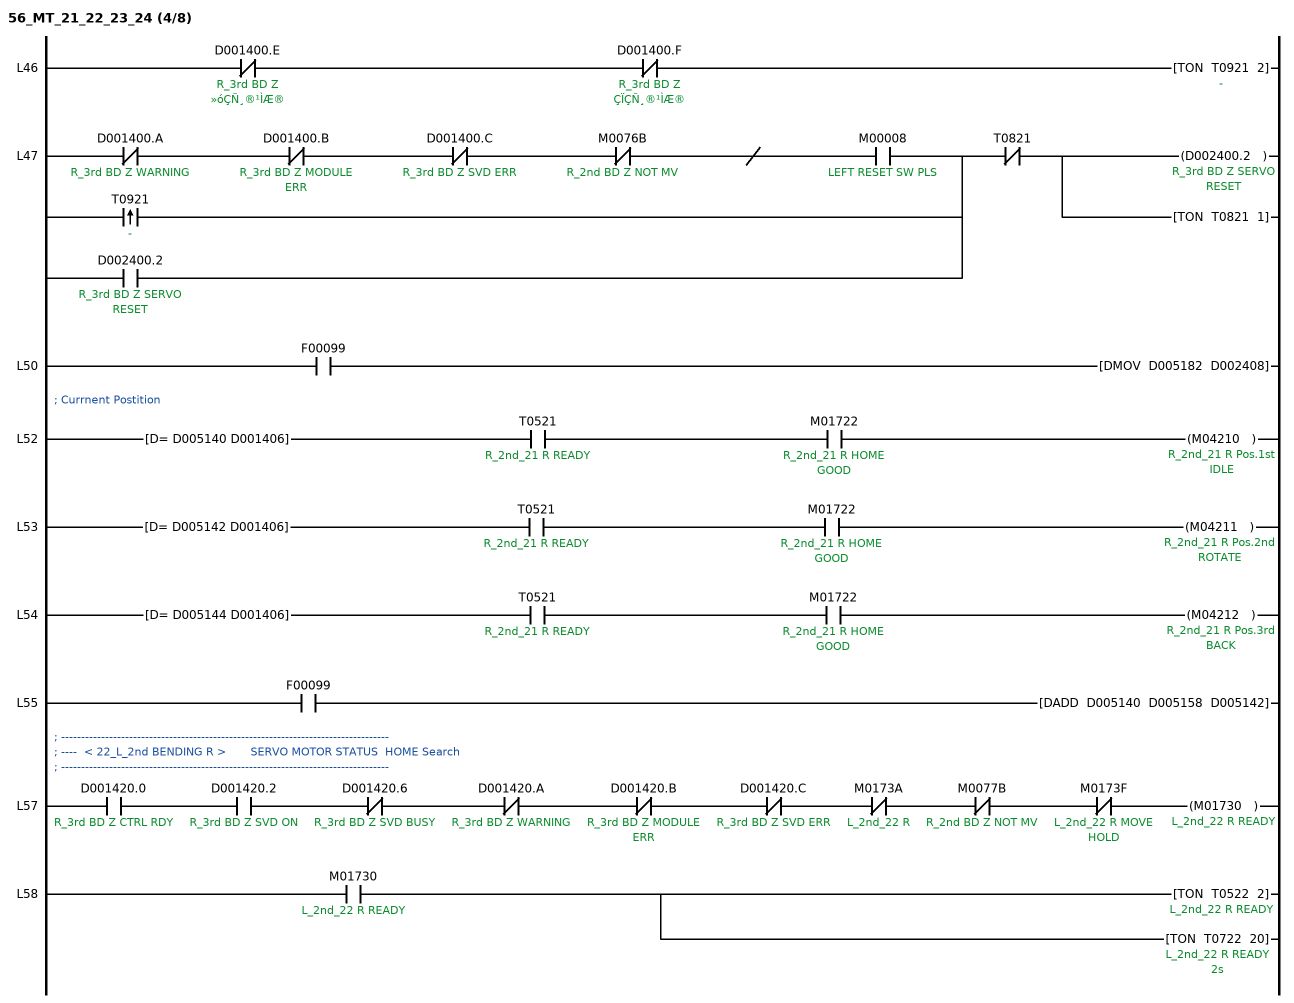
; L46
LOAD NOT  D001400.E	// R_3rd BD Z »óÇÑ¸®¹ÌÆ®
AND NOT   D001400.F	// R_3rd BD Z ÇÏÇÑ¸®¹ÌÆ®
TON       T0921 2	// -
; L47
LOAD NOT  D001400.A	// R_3rd BD Z WARNING
AND NOT   D001400.B	// R_3rd BD Z MODULE ERR
AND NOT   D001400.C	// R_3rd BD Z SVD ERR
AND NOT   M0076B	// R_2nd BD Z NOT MV
NOT
AND       M00008	// LEFT RESET SW PLS
ORP       T0921	// -
OR        D002400.2	// R_3rd BD Z SERVO RESET
AND NOT   T0821
OUT       D002400.2	// R_3rd BD Z SERVO RESET
TON       T0821 1
; L50
LOAD      F00099
DMOV      D005182 D002408
// Currnent Postition
; L52
LOADD=    D005140 D001406
AND       T0521	// R_2nd_21 R READY
AND       M01722	// R_2nd_21 R HOME GOOD
OUT       M04210	// R_2nd_21 R Pos.1st IDLE
; L53
LOADD=    D005142 D001406
AND       T0521	// R_2nd_21 R READY
AND       M01722	// R_2nd_21 R HOME GOOD
OUT       M04211	// R_2nd_21 R Pos.2nd ROTATE
; L54
LOADD=    D005144 D001406
AND       T0521	// R_2nd_21 R READY
AND       M01722	// R_2nd_21 R HOME GOOD
OUT       M04212	// R_2nd_21 R Pos.3rd BACK
; L55
LOAD      F00099
DADD      D005140 D005158 D005142
// ----------------------------------------------------------------------------------
// 
// ----  < 22_L_2nd BENDING R >       SERVO MOTOR STATUS  HOME Search
// 
// ----------------------------------------------------------------------------------
; L57
LOAD      D001420.0	// R_3rd BD Z CTRL RDY
AND       D001420.2	// R_3rd BD Z SVD ON
AND NOT   D001420.6	// R_3rd BD Z SVD BUSY
AND NOT   D001420.A	// R_3rd BD Z WARNING
AND NOT   D001420.B	// R_3rd BD Z MODULE ERR
AND NOT   D001420.C	// R_3rd BD Z SVD ERR
AND NOT   M0173A	// L_2nd_22 R
AND NOT   M0077B	// R_2nd BD Z NOT MV
AND NOT   M0173F	// L_2nd_22 R MOVE HOLD
OUT       M01730	// L_2nd_22 R READY
; L58
LOAD      M01730	// L_2nd_22 R READY
TON       T0522 2	// L_2nd_22 R READY
TON       T0722 20	// L_2nd_22 R READY 2s

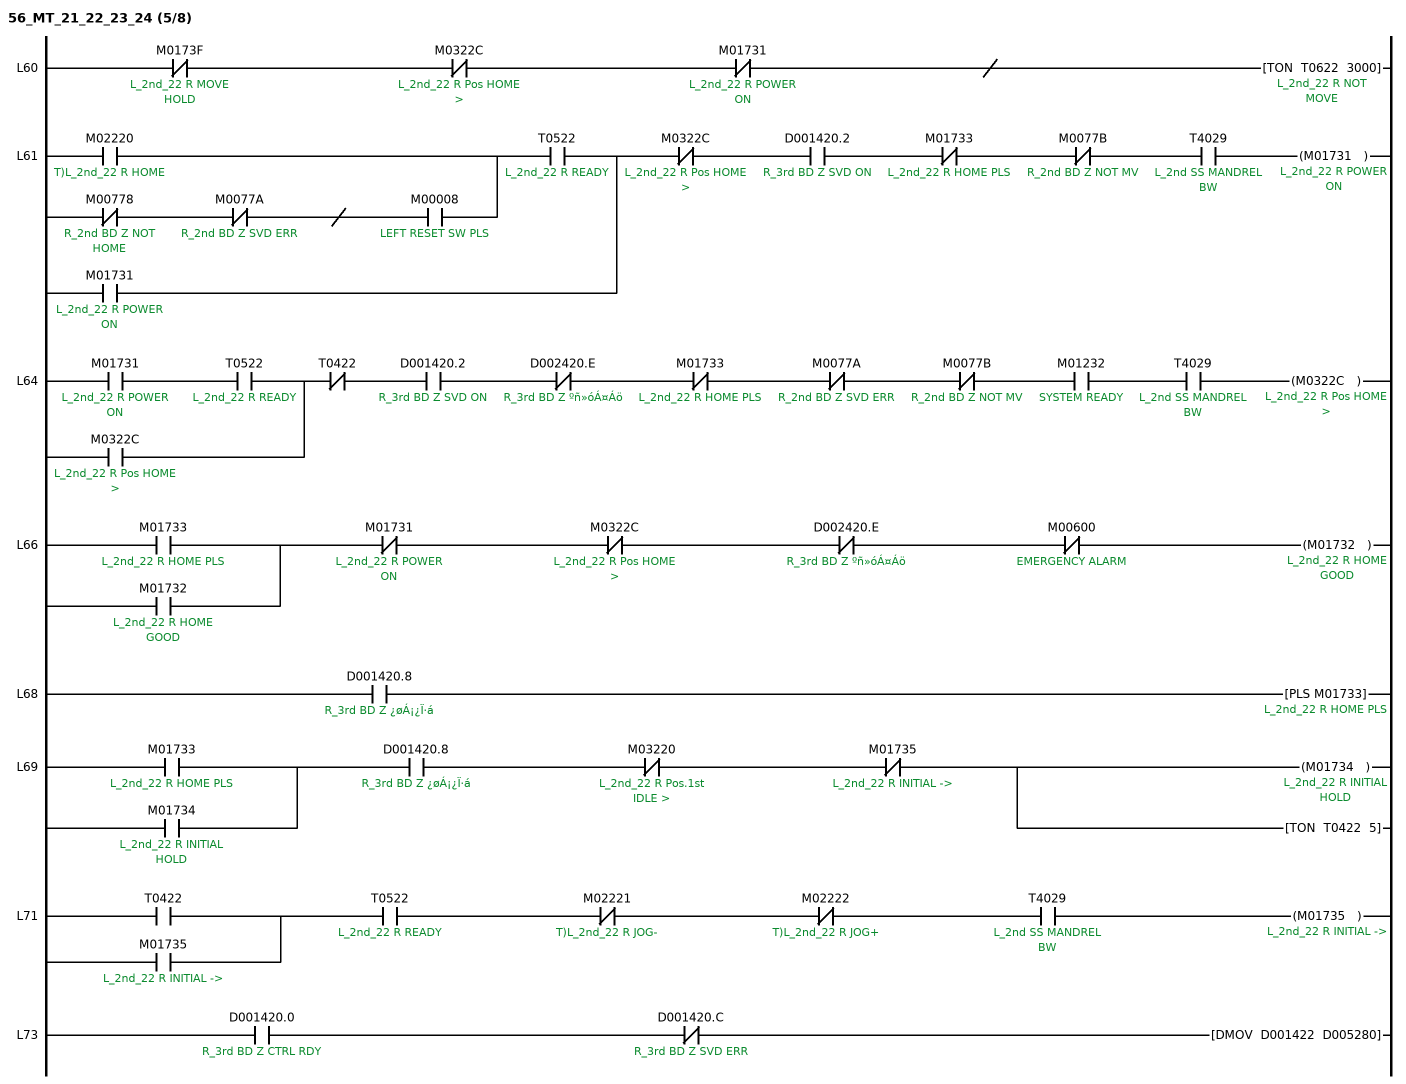
; L60
LOAD NOT  M0173F	// L_2nd_22 R MOVE HOLD
AND NOT   M0322C	// L_2nd_22 R Pos HOME >
AND NOT   M01731	// L_2nd_22 R POWER ON
NOT
TON       T0622 3000	// L_2nd_22 R NOT MOVE
; L61
LOAD      M02220	// T)L_2nd_22 R HOME
LOAD NOT  M00778	// R_2nd BD Z NOT HOME
AND NOT   M0077A	// R_2nd BD Z SVD ERR
NOT
AND       M00008	// LEFT RESET SW PLS
OR LOAD
AND       T0522	// L_2nd_22 R READY
OR        M01731	// L_2nd_22 R POWER ON
AND NOT   M0322C	// L_2nd_22 R Pos HOME >
AND       D001420.2	// R_3rd BD Z SVD ON
AND NOT   M01733	// L_2nd_22 R HOME PLS
AND NOT   M0077B	// R_2nd BD Z NOT MV
AND       T4029	// L_2nd SS MANDREL BW
OUT       M01731	// L_2nd_22 R POWER ON
; L64
LOAD      M01731	// L_2nd_22 R POWER ON
AND       T0522	// L_2nd_22 R READY
OR        M0322C	// L_2nd_22 R Pos HOME >
AND NOT   T0422
AND       D001420.2	// R_3rd BD Z SVD ON
AND NOT   D002420.E	// R_3rd BD Z ºñ»óÁ¤Áö
AND NOT   M01733	// L_2nd_22 R HOME PLS
AND NOT   M0077A	// R_2nd BD Z SVD ERR
AND NOT   M0077B	// R_2nd BD Z NOT MV
AND       M01232	// SYSTEM READY
AND       T4029	// L_2nd SS MANDREL BW
OUT       M0322C	// L_2nd_22 R Pos HOME >
; L66
LOAD      M01733	// L_2nd_22 R HOME PLS
OR        M01732	// L_2nd_22 R HOME GOOD
AND NOT   M01731	// L_2nd_22 R POWER ON
AND NOT   M0322C	// L_2nd_22 R Pos HOME >
AND NOT   D002420.E	// R_3rd BD Z ºñ»óÁ¤Áö
AND NOT   M00600	// EMERGENCY ALARM
OUT       M01732	// L_2nd_22 R HOME GOOD
; L68
LOAD      D001420.8	// R_3rd BD Z ¿øÁ¡¿Ï·á
OUTP      M01733	// L_2nd_22 R HOME PLS
; L69
LOAD      M01733	// L_2nd_22 R HOME PLS
OR        M01734	// L_2nd_22 R INITIAL HOLD
AND       D001420.8	// R_3rd BD Z ¿øÁ¡¿Ï·á
AND NOT   M03220	// L_2nd_22 R Pos.1st IDLE >
AND NOT   M01735	// L_2nd_22 R INITIAL ->
OUT       M01734	// L_2nd_22 R INITIAL HOLD
TON       T0422 5
; L71
LOAD      T0422
OR        M01735	// L_2nd_22 R INITIAL ->
AND       T0522	// L_2nd_22 R READY
AND NOT   M02221	// T)L_2nd_22 R JOG-
AND NOT   M02222	// T)L_2nd_22 R JOG+
AND       T4029	// L_2nd SS MANDREL BW
OUT       M01735	// L_2nd_22 R INITIAL ->
; L73
LOAD      D001420.0	// R_3rd BD Z CTRL RDY
AND NOT   D001420.C	// R_3rd BD Z SVD ERR
DMOV      D001422 D005280

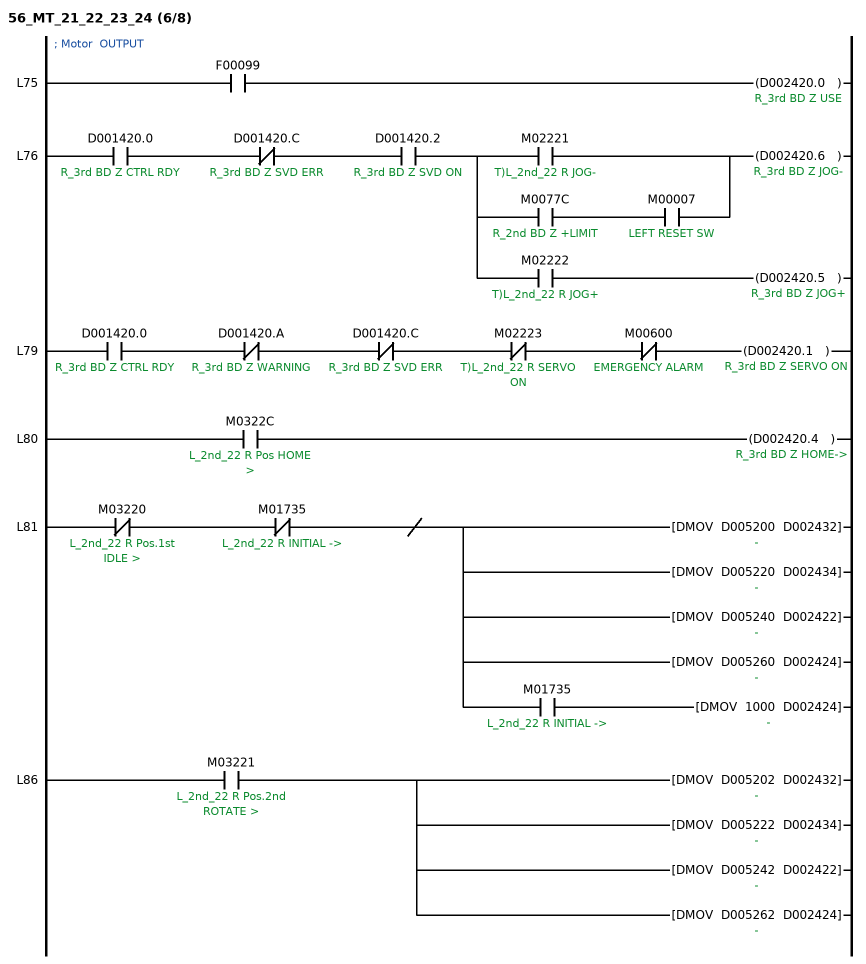
//  Motor  OUTPUT
; L75
LOAD      F00099
OUT       D002420.0	// R_3rd BD Z USE
; L76
LOAD      D001420.0	// R_3rd BD Z CTRL RDY
AND NOT   D001420.C	// R_3rd BD Z SVD ERR
AND       D001420.2	// R_3rd BD Z SVD ON
MPUSH
LOAD      M02221	// T)L_2nd_22 R JOG-
LOAD      M0077C	// R_2nd BD Z +LIMIT
AND       M00007	// LEFT RESET SW
OR LOAD
AND LOAD
OUT       D002420.6	// R_3rd BD Z JOG-
MPOP
AND       M02222	// T)L_2nd_22 R JOG+
OUT       D002420.5	// R_3rd BD Z JOG+
; L79
LOAD      D001420.0	// R_3rd BD Z CTRL RDY
AND NOT   D001420.A	// R_3rd BD Z WARNING
AND NOT   D001420.C	// R_3rd BD Z SVD ERR
AND NOT   M02223	// T)L_2nd_22 R SERVO ON
AND NOT   M00600	// EMERGENCY ALARM
OUT       D002420.1	// R_3rd BD Z SERVO ON
; L80
LOAD      M0322C	// L_2nd_22 R Pos HOME >
OUT       D002420.4	// R_3rd BD Z HOME->
; L81
LOAD NOT  M03220	// L_2nd_22 R Pos.1st IDLE >
AND NOT   M01735	// L_2nd_22 R INITIAL ->
NOT
DMOV      D005200 D002432	// -
DMOV      D005220 D002434	// -
DMOV      D005240 D002422	// -
DMOV      D005260 D002424	// -
AND       M01735	// L_2nd_22 R INITIAL ->
DMOV      1000 D002424	// -
; L86
LOAD      M03221	// L_2nd_22 R Pos.2nd ROTATE >
DMOV      D005202 D002432	// -
DMOV      D005222 D002434	// -
DMOV      D005242 D002422	// -
DMOV      D005262 D002424	// -

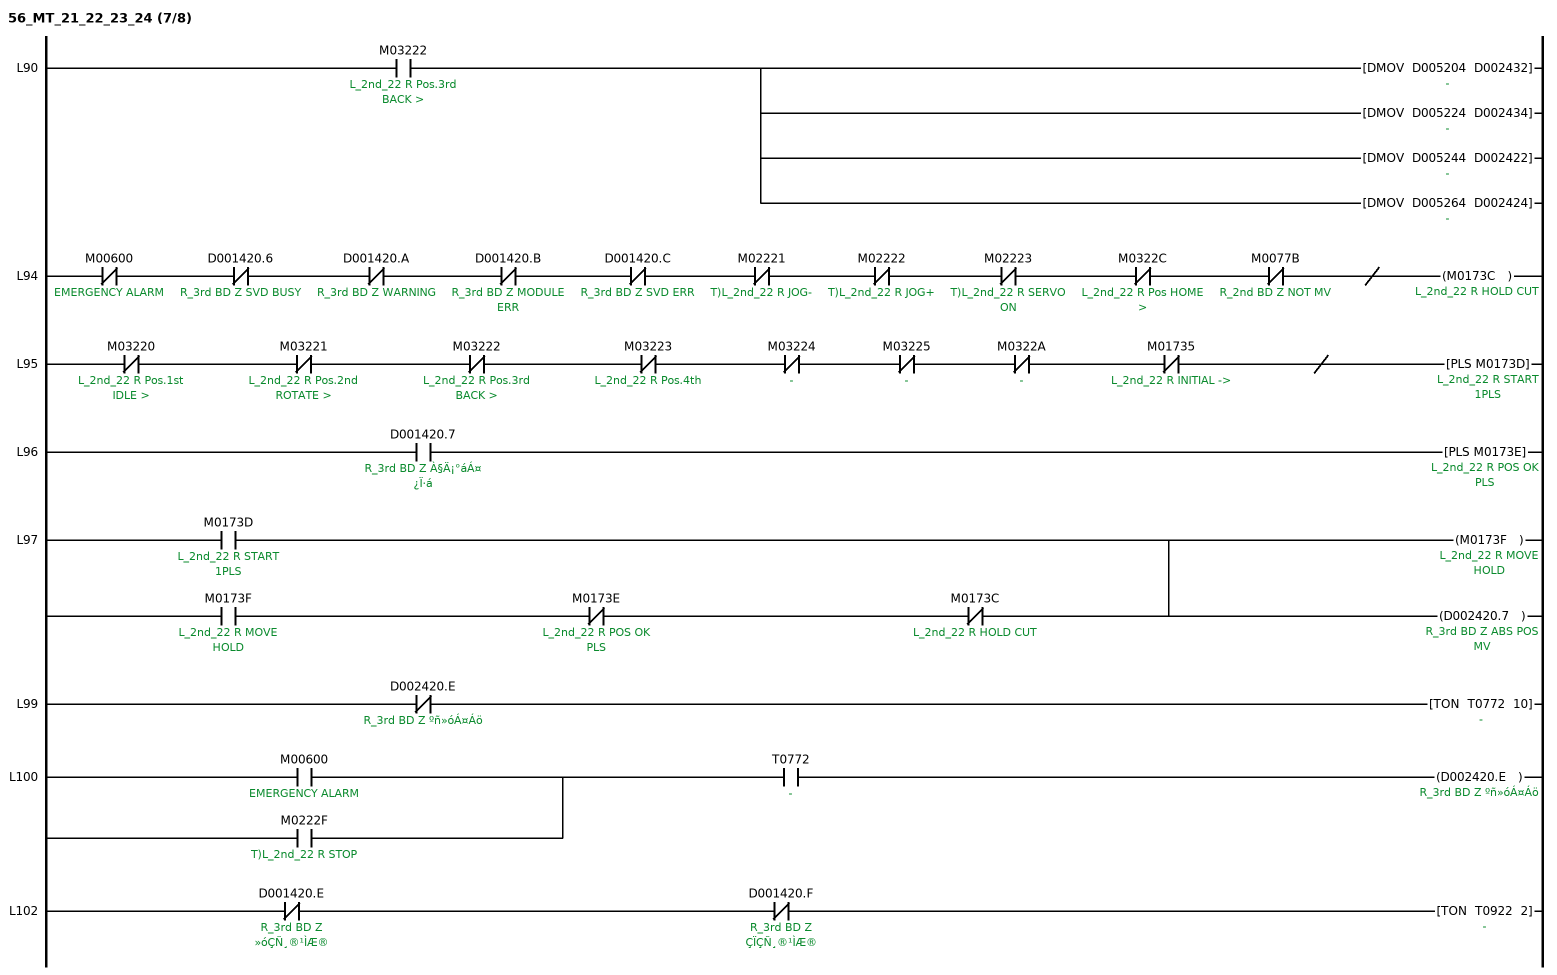
; L90
LOAD      M03222	// L_2nd_22 R Pos.3rd BACK >
DMOV      D005204 D002432	// -
DMOV      D005224 D002434	// -
DMOV      D005244 D002422	// -
DMOV      D005264 D002424	// -
; L94
LOAD NOT  M00600	// EMERGENCY ALARM
AND NOT   D001420.6	// R_3rd BD Z SVD BUSY
AND NOT   D001420.A	// R_3rd BD Z WARNING
AND NOT   D001420.B	// R_3rd BD Z MODULE ERR
AND NOT   D001420.C	// R_3rd BD Z SVD ERR
AND NOT   M02221	// T)L_2nd_22 R JOG-
AND NOT   M02222	// T)L_2nd_22 R JOG+
AND NOT   M02223	// T)L_2nd_22 R SERVO ON
AND NOT   M0322C	// L_2nd_22 R Pos HOME >
AND NOT   M0077B	// R_2nd BD Z NOT MV
NOT
OUT       M0173C	// L_2nd_22 R HOLD CUT
; L95
LOAD NOT  M03220	// L_2nd_22 R Pos.1st IDLE >
AND NOT   M03221	// L_2nd_22 R Pos.2nd ROTATE >
AND NOT   M03222	// L_2nd_22 R Pos.3rd BACK >
AND NOT   M03223	// L_2nd_22 R Pos.4th 
AND NOT   M03224	// -
AND NOT   M03225	// -
AND NOT   M0322A	// -
AND NOT   M01735	// L_2nd_22 R INITIAL ->
NOT
OUTP      M0173D	// L_2nd_22 R START 1PLS
; L96
LOAD      D001420.7	// R_3rd BD Z À§Ä¡°áÁ¤ ¿Ï·á
OUTP      M0173E	// L_2nd_22 R POS OK PLS
; L97
LOAD      M0173D	// L_2nd_22 R START 1PLS
LOAD      M0173F	// L_2nd_22 R MOVE HOLD
AND NOT   M0173E	// L_2nd_22 R POS OK PLS
AND NOT   M0173C	// L_2nd_22 R HOLD CUT
OR LOAD
OUT       M0173F	// L_2nd_22 R MOVE HOLD
OUT       D002420.7	// R_3rd BD Z ABS POS MV
; L99
LOAD NOT  D002420.E	// R_3rd BD Z ºñ»óÁ¤Áö
TON       T0772 10	// -
; L100
LOAD      M00600	// EMERGENCY ALARM
OR        M0222F	// T)L_2nd_22 R STOP
AND       T0772	// -
OUT       D002420.E	// R_3rd BD Z ºñ»óÁ¤Áö
; L102
LOAD NOT  D001420.E	// R_3rd BD Z »óÇÑ¸®¹ÌÆ®
AND NOT   D001420.F	// R_3rd BD Z ÇÏÇÑ¸®¹ÌÆ®
TON       T0922 2	// -

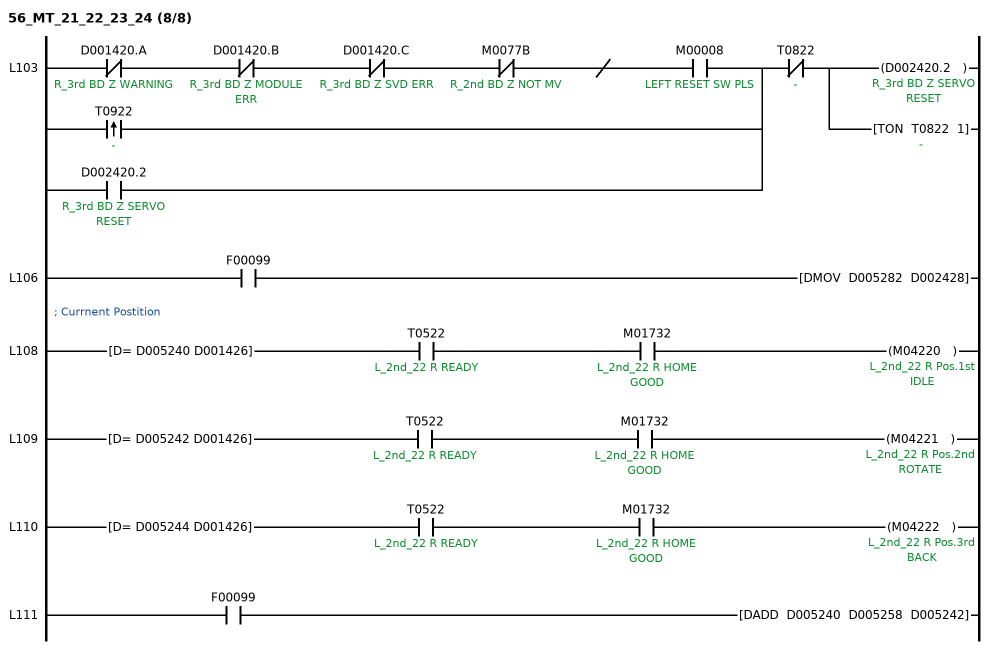
; L103
LOAD NOT  D001420.A	// R_3rd BD Z WARNING
AND NOT   D001420.B	// R_3rd BD Z MODULE ERR
AND NOT   D001420.C	// R_3rd BD Z SVD ERR
AND NOT   M0077B	// R_2nd BD Z NOT MV
NOT
AND       M00008	// LEFT RESET SW PLS
ORP       T0922	// -
OR        D002420.2	// R_3rd BD Z SERVO RESET
AND NOT   T0822	// -
OUT       D002420.2	// R_3rd BD Z SERVO RESET
TON       T0822 1	// -
; L106
LOAD      F00099
DMOV      D005282 D002428
// Currnent Postition
; L108
LOADD=    D005240 D001426
AND       T0522	// L_2nd_22 R READY
AND       M01732	// L_2nd_22 R HOME GOOD
OUT       M04220	// L_2nd_22 R Pos.1st IDLE
; L109
LOADD=    D005242 D001426
AND       T0522	// L_2nd_22 R READY
AND       M01732	// L_2nd_22 R HOME GOOD
OUT       M04221	// L_2nd_22 R Pos.2nd ROTATE
; L110
LOADD=    D005244 D001426
AND       T0522	// L_2nd_22 R READY
AND       M01732	// L_2nd_22 R HOME GOOD
OUT       M04222	// L_2nd_22 R Pos.3rd BACK
; L111
LOAD      F00099
DADD      D005240 D005258 D005242

PROGRAM 81_OUTPUT (task: ½ºÄµ ÇÁ·Î±×·¥)

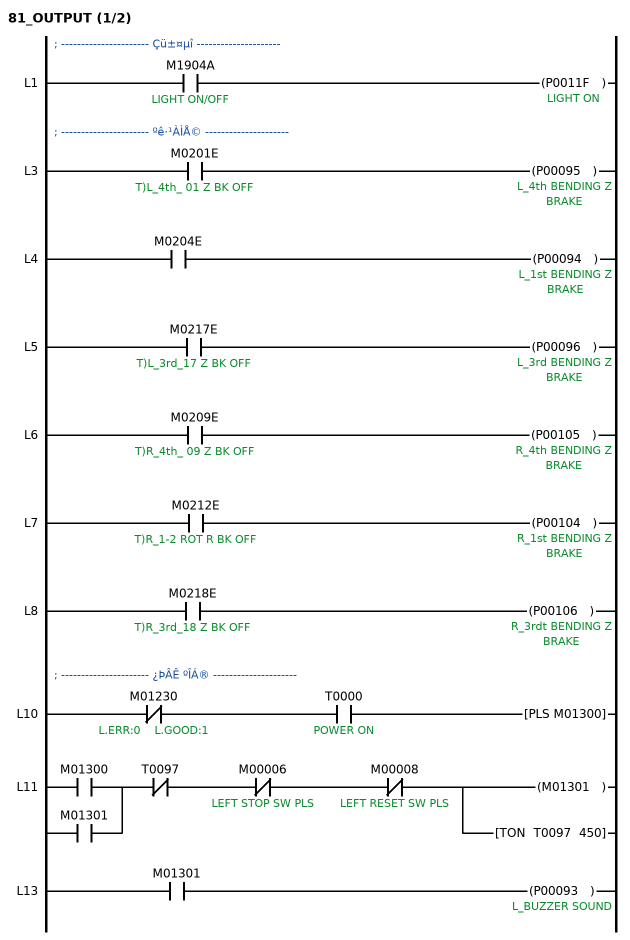
// ---------------------- Çü±¤µî ---------------------
; L1
LOAD      M1904A	// LIGHT ON/OFF
OUT       P0011F	// LIGHT ON
// ---------------------- ºê·¹ÀÌÅ© ---------------------
; L3
LOAD      M0201E	// T)L_4th_ 01 Z BK OFF
OUT       P00095	// L_4th BENDING Z BRAKE
; L4
LOAD      M0204E
OUT       P00094	// L_1st BENDING Z BRAKE
; L5
LOAD      M0217E	// T)L_3rd_17 Z BK OFF
OUT       P00096	// L_3rd BENDING Z BRAKE
; L6
LOAD      M0209E	// T)R_4th_ 09 Z BK OFF
OUT       P00105	// R_4th BENDING Z BRAKE
; L7
LOAD      M0212E	// T)R_1-2 ROT R BK OFF
OUT       P00104	// R_1st BENDING Z BRAKE
; L8
LOAD      M0218E	// T)R_3rd_18 Z BK OFF
OUT       P00106	// R_3rdt BENDING Z BRAKE
// ---------------------- ¿ÞÂÊ ºÎÁ® ---------------------
; L10
LOAD NOT  M01230	// L.ERR:0    L.GOOD:1
AND       T0000	// POWER ON
OUTP      M01300
; L11
LOAD      M01300
OR        M01301
AND NOT   T0097
AND NOT   M00006	// LEFT STOP SW PLS
AND NOT   M00008	// LEFT RESET SW PLS
OUT       M01301
TON       T0097 450
; L13
LOAD      M01301
OUT       P00093	// L_BUZZER SOUND

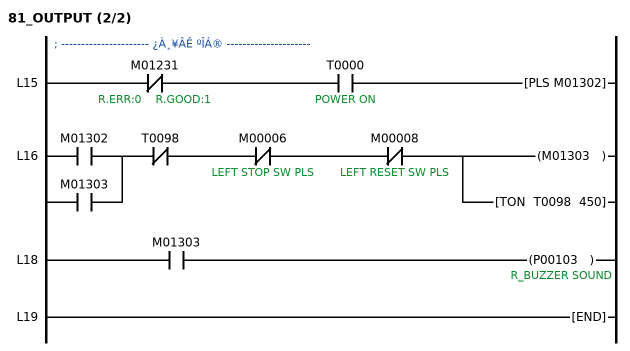
// ---------------------- ¿À¸¥ÂÊ ºÎÁ® ---------------------
; L15
LOAD NOT  M01231	// R.ERR:0    R.GOOD:1
AND       T0000	// POWER ON
OUTP      M01302
; L16
LOAD      M01302
OR        M01303
AND NOT   T0098
AND NOT   M00006	// LEFT STOP SW PLS
AND NOT   M00008	// LEFT RESET SW PLS
OUT       M01303
TON       T0098 450
; L18
LOAD      M01303
OUT       P00103	// R_BUZZER SOUND
; L19
END

PROGRAM 82_L_MANUAL (task: ½ºÄµ ÇÁ·Î±×·¥)

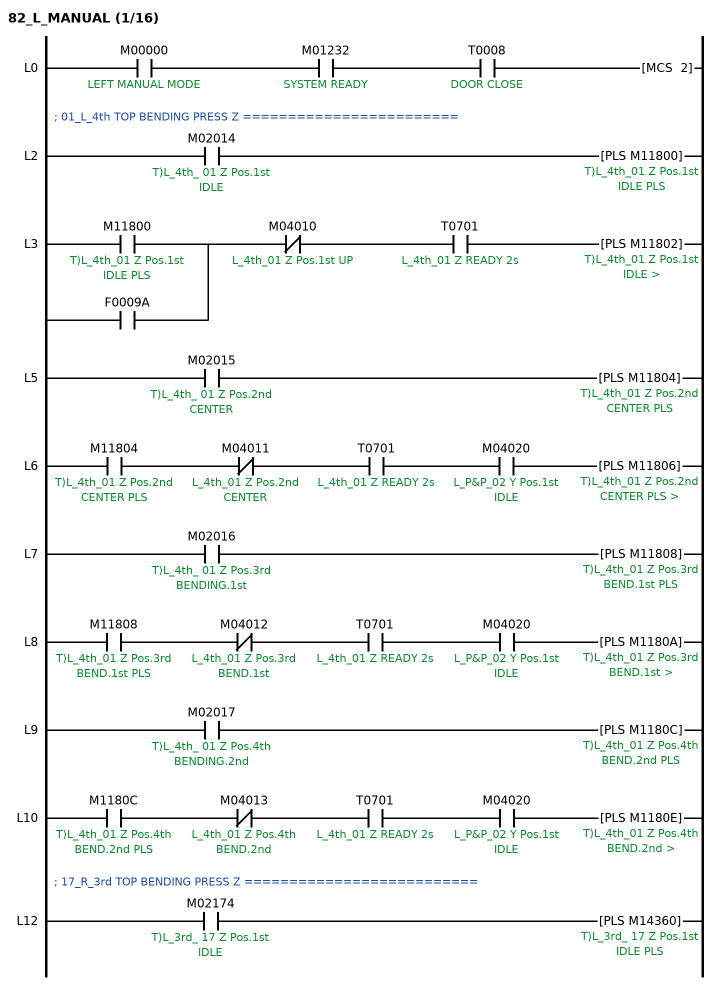
; L0
LOAD      M00000	// LEFT MANUAL MODE
AND       M01232	// SYSTEM READY
AND       T0008	// DOOR CLOSE
MCS       2
// 01_L_4th TOP BENDING PRESS Z ======================== 
; L2
LOAD      M02014	// T)L_4th_ 01 Z Pos.1st IDLE
OUTP      M11800	// T)L_4th_01 Z Pos.1st IDLE PLS
; L3
LOAD      M11800	// T)L_4th_01 Z Pos.1st IDLE PLS
OR        F0009A
AND NOT   M04010	// L_4th_01 Z Pos.1st UP
AND       T0701	// L_4th_01 Z READY 2s
OUTP      M11802	// T)L_4th_01 Z Pos.1st IDLE >
; L5
LOAD      M02015	// T)L_4th_ 01 Z Pos.2nd CENTER
OUTP      M11804	// T)L_4th_01 Z Pos.2nd CENTER PLS
; L6
LOAD      M11804	// T)L_4th_01 Z Pos.2nd CENTER PLS
AND NOT   M04011	// L_4th_01 Z Pos.2nd CENTER
AND       T0701	// L_4th_01 Z READY 2s
AND       M04020	// L_P&P_02 Y Pos.1st IDLE
OUTP      M11806	// T)L_4th_01 Z Pos.2nd CENTER PLS >
; L7
LOAD      M02016	// T)L_4th_ 01 Z Pos.3rd BENDING.1st
OUTP      M11808	// T)L_4th_01 Z Pos.3rd BEND.1st PLS
; L8
LOAD      M11808	// T)L_4th_01 Z Pos.3rd BEND.1st PLS
AND NOT   M04012	// L_4th_01 Z Pos.3rd BEND.1st
AND       T0701	// L_4th_01 Z READY 2s
AND       M04020	// L_P&P_02 Y Pos.1st IDLE
OUTP      M1180A	// T)L_4th_01 Z Pos.3rd BEND.1st >
; L9
LOAD      M02017	// T)L_4th_ 01 Z Pos.4th BENDING.2nd
OUTP      M1180C	// T)L_4th_01 Z Pos.4th BEND.2nd PLS
; L10
LOAD      M1180C	// T)L_4th_01 Z Pos.4th BEND.2nd PLS
AND NOT   M04013	// L_4th_01 Z Pos.4th BEND.2nd
AND       T0701	// L_4th_01 Z READY 2s
AND       M04020	// L_P&P_02 Y Pos.1st IDLE
OUTP      M1180E	// T)L_4th_01 Z Pos.4th BEND.2nd >
// 17_R_3rd TOP BENDING PRESS Z ==========================
; L12
LOAD      M02174	// T)L_3rd_ 17 Z Pos.1st IDLE
OUTP      M14360	// T)L_3rd_ 17 Z Pos.1st IDLE PLS

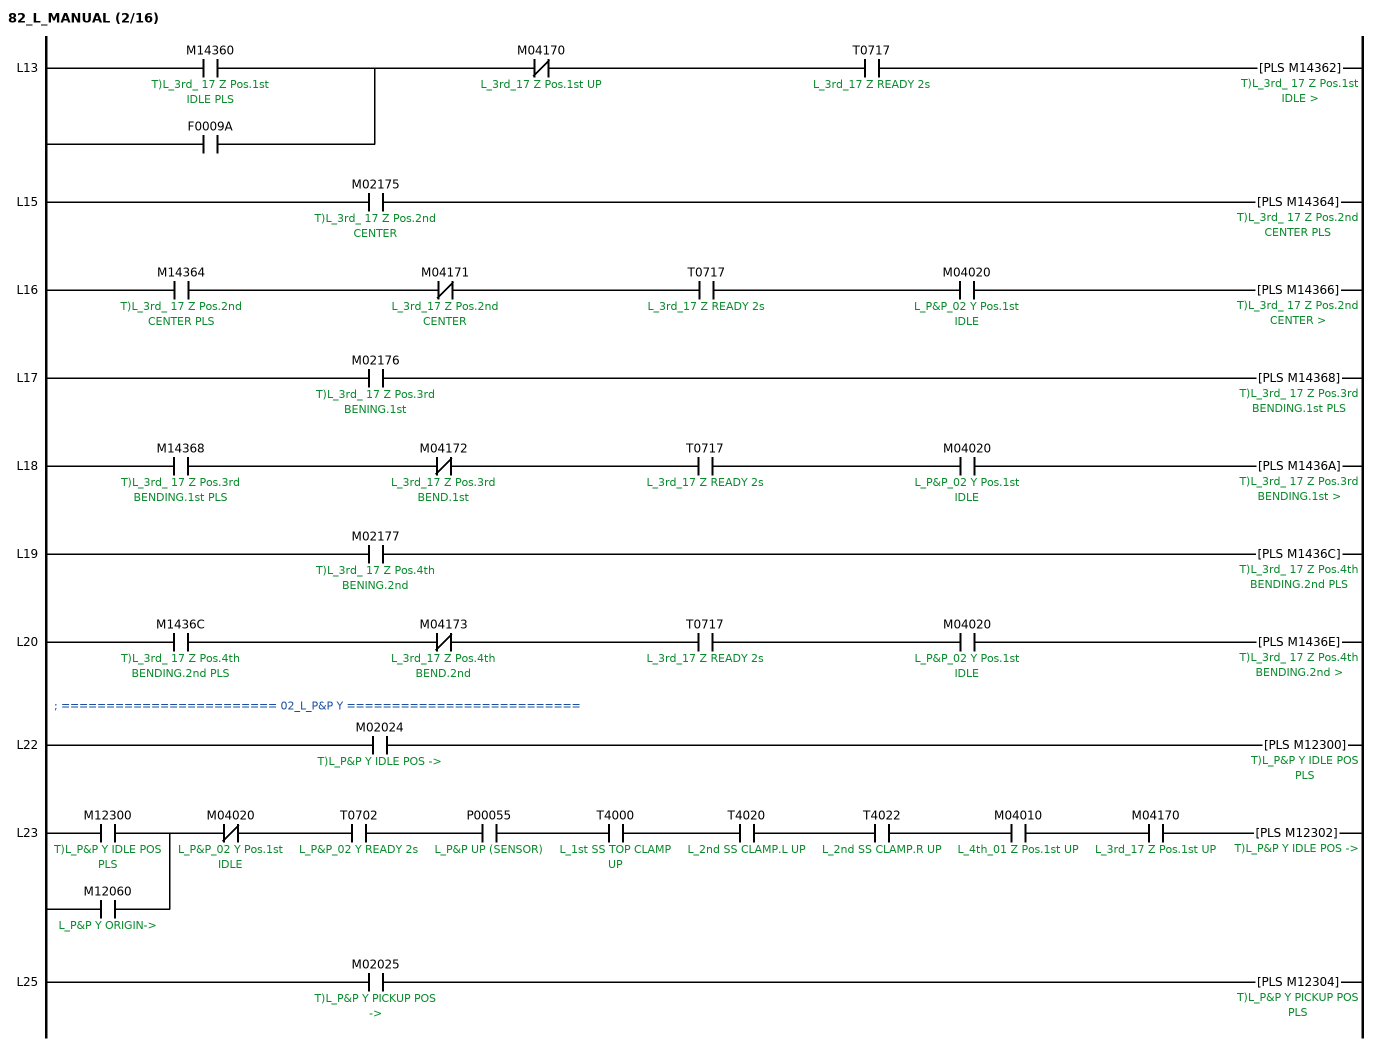
; L13
LOAD      M14360	// T)L_3rd_ 17 Z Pos.1st IDLE PLS
OR        F0009A
AND NOT   M04170	// L_3rd_17 Z Pos.1st UP
AND       T0717	// L_3rd_17 Z READY 2s
OUTP      M14362	// T)L_3rd_ 17 Z Pos.1st IDLE >
; L15
LOAD      M02175	// T)L_3rd_ 17 Z Pos.2nd CENTER
OUTP      M14364	// T)L_3rd_ 17 Z Pos.2nd CENTER PLS
; L16
LOAD      M14364	// T)L_3rd_ 17 Z Pos.2nd CENTER PLS
AND NOT   M04171	// L_3rd_17 Z Pos.2nd CENTER
AND       T0717	// L_3rd_17 Z READY 2s
AND       M04020	// L_P&P_02 Y Pos.1st IDLE
OUTP      M14366	// T)L_3rd_ 17 Z Pos.2nd CENTER >
; L17
LOAD      M02176	// T)L_3rd_ 17 Z Pos.3rd BENING.1st
OUTP      M14368	// T)L_3rd_ 17 Z Pos.3rd BENDING.1st PLS
; L18
LOAD      M14368	// T)L_3rd_ 17 Z Pos.3rd BENDING.1st PLS
AND NOT   M04172	// L_3rd_17 Z Pos.3rd BEND.1st
AND       T0717	// L_3rd_17 Z READY 2s
AND       M04020	// L_P&P_02 Y Pos.1st IDLE
OUTP      M1436A	// T)L_3rd_ 17 Z Pos.3rd BENDING.1st >
; L19
LOAD      M02177	// T)L_3rd_ 17 Z Pos.4th BENING.2nd
OUTP      M1436C	// T)L_3rd_ 17 Z Pos.4th BENDING.2nd PLS
; L20
LOAD      M1436C	// T)L_3rd_ 17 Z Pos.4th BENDING.2nd PLS
AND NOT   M04173	// L_3rd_17 Z Pos.4th BEND.2nd
AND       T0717	// L_3rd_17 Z READY 2s
AND       M04020	// L_P&P_02 Y Pos.1st IDLE
OUTP      M1436E	// T)L_3rd_ 17 Z Pos.4th BENDING.2nd >
// ======================== 02_L_P&P Y ==========================
; L22
LOAD      M02024	// T)L_P&P Y IDLE POS ->
OUTP      M12300	// T)L_P&P Y IDLE POS PLS
; L23
LOAD      M12300	// T)L_P&P Y IDLE POS PLS
OR        M12060	// L_P&P Y ORIGIN->
AND NOT   M04020	// L_P&P_02 Y Pos.1st IDLE
AND       T0702	// L_P&P_02 Y READY 2s
AND       P00055	// L_P&P UP (SENSOR)
AND       T4000	// L_1st SS TOP CLAMP    UP
AND       T4020	// L_2nd SS CLAMP.L UP
AND       T4022	// L_2nd SS CLAMP.R UP
AND       M04010	// L_4th_01 Z Pos.1st UP
AND       M04170	// L_3rd_17 Z Pos.1st UP
OUTP      M12302	// T)L_P&P Y IDLE POS ->
; L25
LOAD      M02025	// T)L_P&P Y PICKUP POS ->
OUTP      M12304	// T)L_P&P Y PICKUP POS PLS

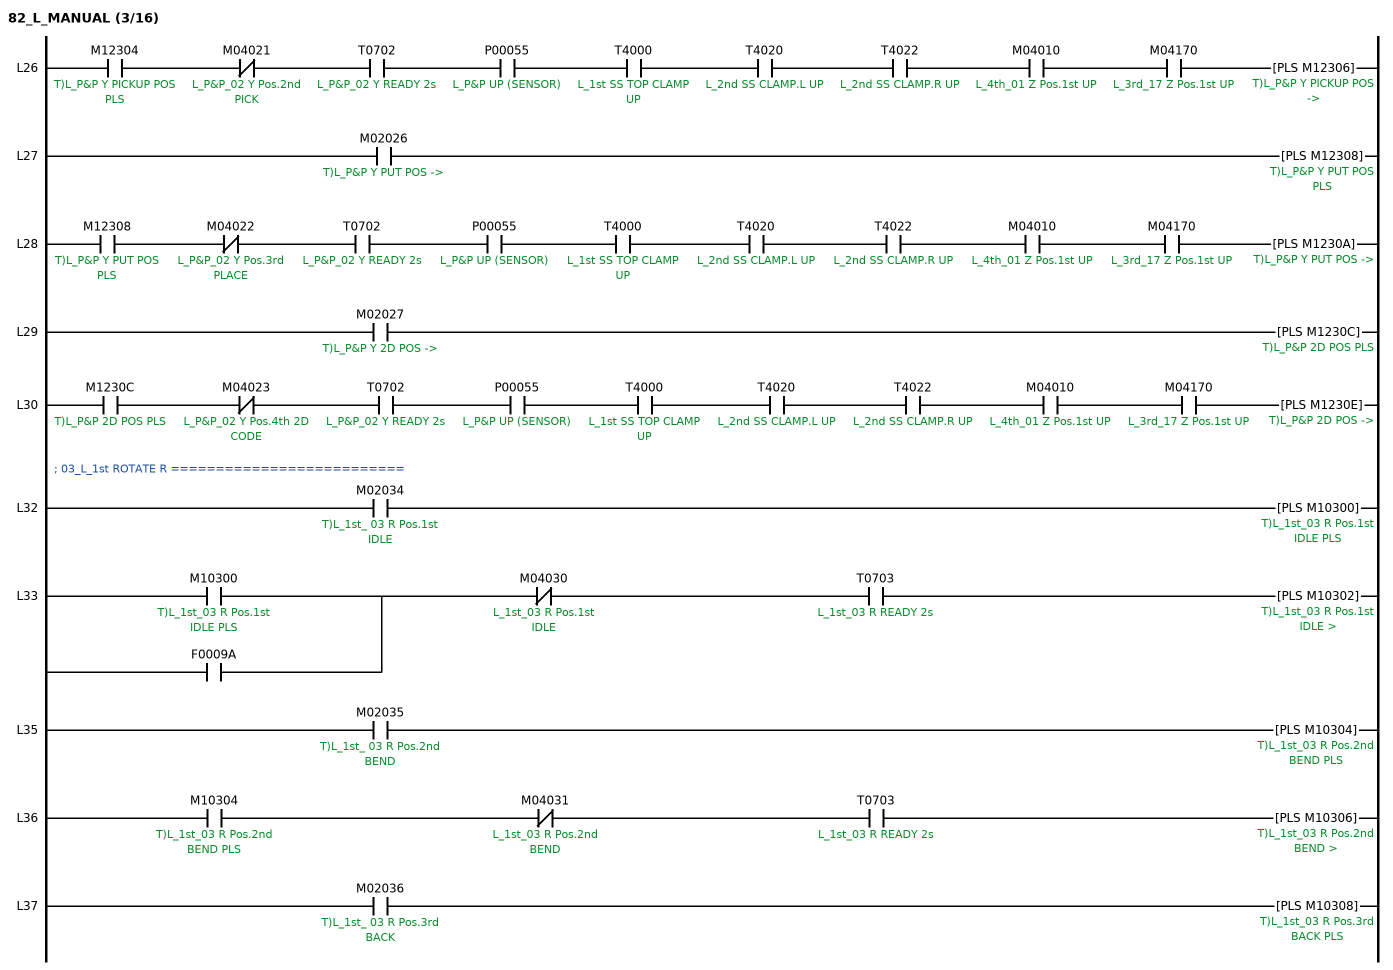
; L26
LOAD      M12304	// T)L_P&P Y PICKUP POS PLS
AND NOT   M04021	// L_P&P_02 Y Pos.2nd PICK
AND       T0702	// L_P&P_02 Y READY 2s
AND       P00055	// L_P&P UP (SENSOR)
AND       T4000	// L_1st SS TOP CLAMP    UP
AND       T4020	// L_2nd SS CLAMP.L UP
AND       T4022	// L_2nd SS CLAMP.R UP
AND       M04010	// L_4th_01 Z Pos.1st UP
AND       M04170	// L_3rd_17 Z Pos.1st UP
OUTP      M12306	// T)L_P&P Y PICKUP POS ->
; L27
LOAD      M02026	// T)L_P&P Y PUT POS ->
OUTP      M12308	// T)L_P&P Y PUT POS PLS
; L28
LOAD      M12308	// T)L_P&P Y PUT POS PLS
AND NOT   M04022	// L_P&P_02 Y Pos.3rd PLACE
AND       T0702	// L_P&P_02 Y READY 2s
AND       P00055	// L_P&P UP (SENSOR)
AND       T4000	// L_1st SS TOP CLAMP    UP
AND       T4020	// L_2nd SS CLAMP.L UP
AND       T4022	// L_2nd SS CLAMP.R UP
AND       M04010	// L_4th_01 Z Pos.1st UP
AND       M04170	// L_3rd_17 Z Pos.1st UP
OUTP      M1230A	// T)L_P&P Y PUT POS ->
; L29
LOAD      M02027	// T)L_P&P Y 2D POS ->
OUTP      M1230C	// T)L_P&P 2D POS PLS
; L30
LOAD      M1230C	// T)L_P&P 2D POS PLS
AND NOT   M04023	// L_P&P_02 Y Pos.4th 2D CODE
AND       T0702	// L_P&P_02 Y READY 2s
AND       P00055	// L_P&P UP (SENSOR)
AND       T4000	// L_1st SS TOP CLAMP    UP
AND       T4020	// L_2nd SS CLAMP.L UP
AND       T4022	// L_2nd SS CLAMP.R UP
AND       M04010	// L_4th_01 Z Pos.1st UP
AND       M04170	// L_3rd_17 Z Pos.1st UP
OUTP      M1230E	// T)L_P&P 2D POS ->
// 03_L_1st ROTATE R ==========================
; L32
LOAD      M02034	// T)L_1st_ 03 R Pos.1st IDLE
OUTP      M10300	// T)L_1st_03 R Pos.1st IDLE PLS
; L33
LOAD      M10300	// T)L_1st_03 R Pos.1st IDLE PLS
OR        F0009A
AND NOT   M04030	// L_1st_03 R Pos.1st IDLE
AND       T0703	// L_1st_03 R READY 2s
OUTP      M10302	// T)L_1st_03 R Pos.1st IDLE >
; L35
LOAD      M02035	// T)L_1st_ 03 R Pos.2nd BEND
OUTP      M10304	// T)L_1st_03 R Pos.2nd BEND PLS
; L36
LOAD      M10304	// T)L_1st_03 R Pos.2nd BEND PLS
AND NOT   M04031	// L_1st_03 R Pos.2nd BEND
AND       T0703	// L_1st_03 R READY 2s
OUTP      M10306	// T)L_1st_03 R Pos.2nd BEND >
; L37
LOAD      M02036	// T)L_1st_ 03 R Pos.3rd BACK
OUTP      M10308	// T)L_1st_03 R Pos.3rd BACK PLS

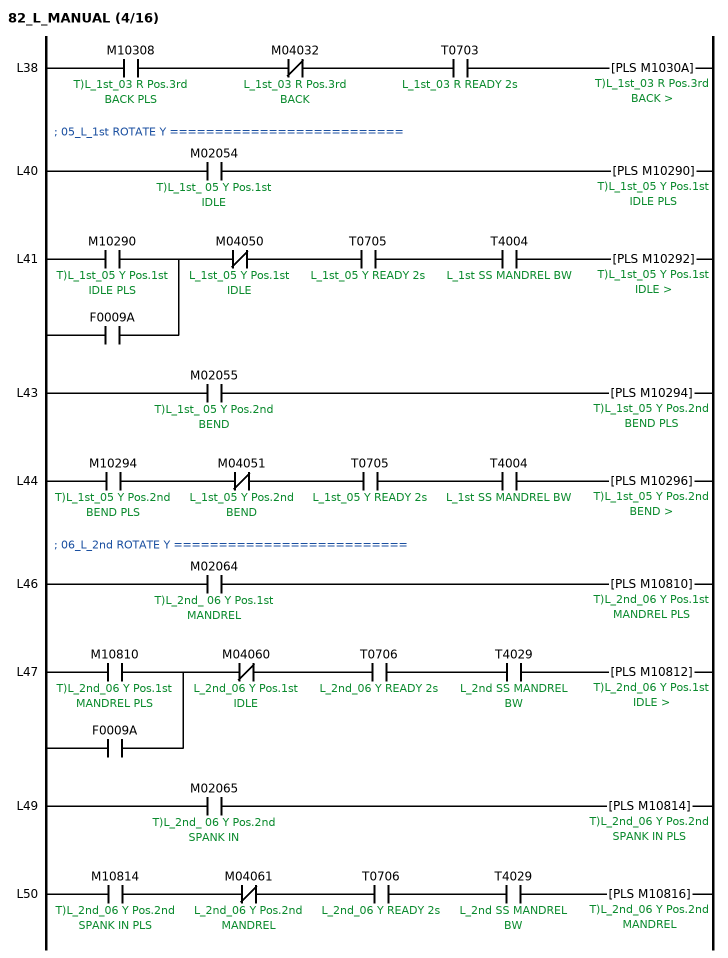
; L38
LOAD      M10308	// T)L_1st_03 R Pos.3rd BACK PLS
AND NOT   M04032	// L_1st_03 R Pos.3rd BACK
AND       T0703	// L_1st_03 R READY 2s
OUTP      M1030A	// T)L_1st_03 R Pos.3rd BACK >
// 05_L_1st ROTATE Y ==========================
; L40
LOAD      M02054	// T)L_1st_ 05 Y Pos.1st IDLE
OUTP      M10290	// T)L_1st_05 Y Pos.1st IDLE PLS
; L41
LOAD      M10290	// T)L_1st_05 Y Pos.1st IDLE PLS
OR        F0009A
AND NOT   M04050	// L_1st_05 Y Pos.1st IDLE
AND       T0705	// L_1st_05 Y READY 2s
AND       T4004	// L_1st SS MANDREL BW
OUTP      M10292	// T)L_1st_05 Y Pos.1st IDLE >
; L43
LOAD      M02055	// T)L_1st_ 05 Y Pos.2nd BEND
OUTP      M10294	// T)L_1st_05 Y Pos.2nd BEND PLS
; L44
LOAD      M10294	// T)L_1st_05 Y Pos.2nd BEND PLS
AND NOT   M04051	// L_1st_05 Y Pos.2nd BEND
AND       T0705	// L_1st_05 Y READY 2s
AND       T4004	// L_1st SS MANDREL BW
OUTP      M10296	// T)L_1st_05 Y Pos.2nd BEND >
// 06_L_2nd ROTATE Y ==========================
; L46
LOAD      M02064	// T)L_2nd_ 06 Y Pos.1st MANDREL
OUTP      M10810	// T)L_2nd_06 Y Pos.1st MANDREL PLS
; L47
LOAD      M10810	// T)L_2nd_06 Y Pos.1st MANDREL PLS
OR        F0009A
AND NOT   M04060	// L_2nd_06 Y Pos.1st IDLE
AND       T0706	// L_2nd_06 Y READY 2s
AND       T4029	// L_2nd SS MANDREL BW
OUTP      M10812	// T)L_2nd_06 Y Pos.1st IDLE >
; L49
LOAD      M02065	// T)L_2nd_ 06 Y Pos.2nd SPANK IN
OUTP      M10814	// T)L_2nd_06 Y Pos.2nd SPANK IN PLS
; L50
LOAD      M10814	// T)L_2nd_06 Y Pos.2nd SPANK IN PLS
AND NOT   M04061	// L_2nd_06 Y Pos.2nd MANDREL
AND       T0706	// L_2nd_06 Y READY 2s
AND       T4029	// L_2nd SS MANDREL BW
OUTP      M10816	// T)L_2nd_06 Y Pos.2nd MANDREL

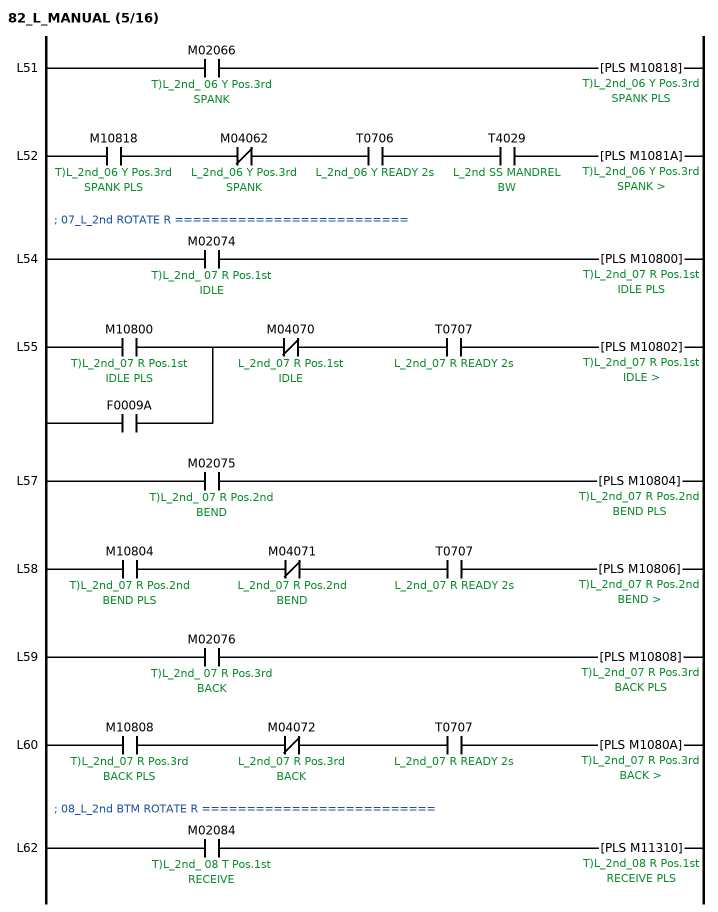
; L51
LOAD      M02066	// T)L_2nd_ 06 Y Pos.3rd SPANK
OUTP      M10818	// T)L_2nd_06 Y Pos.3rd SPANK PLS
; L52
LOAD      M10818	// T)L_2nd_06 Y Pos.3rd SPANK PLS
AND NOT   M04062	// L_2nd_06 Y Pos.3rd SPANK
AND       T0706	// L_2nd_06 Y READY 2s
AND       T4029	// L_2nd SS MANDREL BW
OUTP      M1081A	// T)L_2nd_06 Y Pos.3rd SPANK >
// 07_L_2nd ROTATE R ==========================
; L54
LOAD      M02074	// T)L_2nd_ 07 R Pos.1st IDLE
OUTP      M10800	// T)L_2nd_07 R Pos.1st IDLE PLS
; L55
LOAD      M10800	// T)L_2nd_07 R Pos.1st IDLE PLS
OR        F0009A
AND NOT   M04070	// L_2nd_07 R Pos.1st IDLE
AND       T0707	// L_2nd_07 R READY 2s
OUTP      M10802	// T)L_2nd_07 R Pos.1st IDLE >
; L57
LOAD      M02075	// T)L_2nd_ 07 R Pos.2nd BEND
OUTP      M10804	// T)L_2nd_07 R Pos.2nd BEND PLS
; L58
LOAD      M10804	// T)L_2nd_07 R Pos.2nd BEND PLS
AND NOT   M04071	// L_2nd_07 R Pos.2nd BEND
AND       T0707	// L_2nd_07 R READY 2s
OUTP      M10806	// T)L_2nd_07 R Pos.2nd BEND >
; L59
LOAD      M02076	// T)L_2nd_ 07 R Pos.3rd BACK
OUTP      M10808	// T)L_2nd_07 R Pos.3rd BACK PLS
; L60
LOAD      M10808	// T)L_2nd_07 R Pos.3rd BACK PLS
AND NOT   M04072	// L_2nd_07 R Pos.3rd BACK
AND       T0707	// L_2nd_07 R READY 2s
OUTP      M1080A	// T)L_2nd_07 R Pos.3rd BACK >
// 08_L_2nd BTM ROTATE R ==========================
; L62
LOAD      M02084	// T)L_2nd_ 08 T Pos.1st RECEIVE
OUTP      M11310	// T)L_2nd_08 R Pos.1st RECEIVE PLS

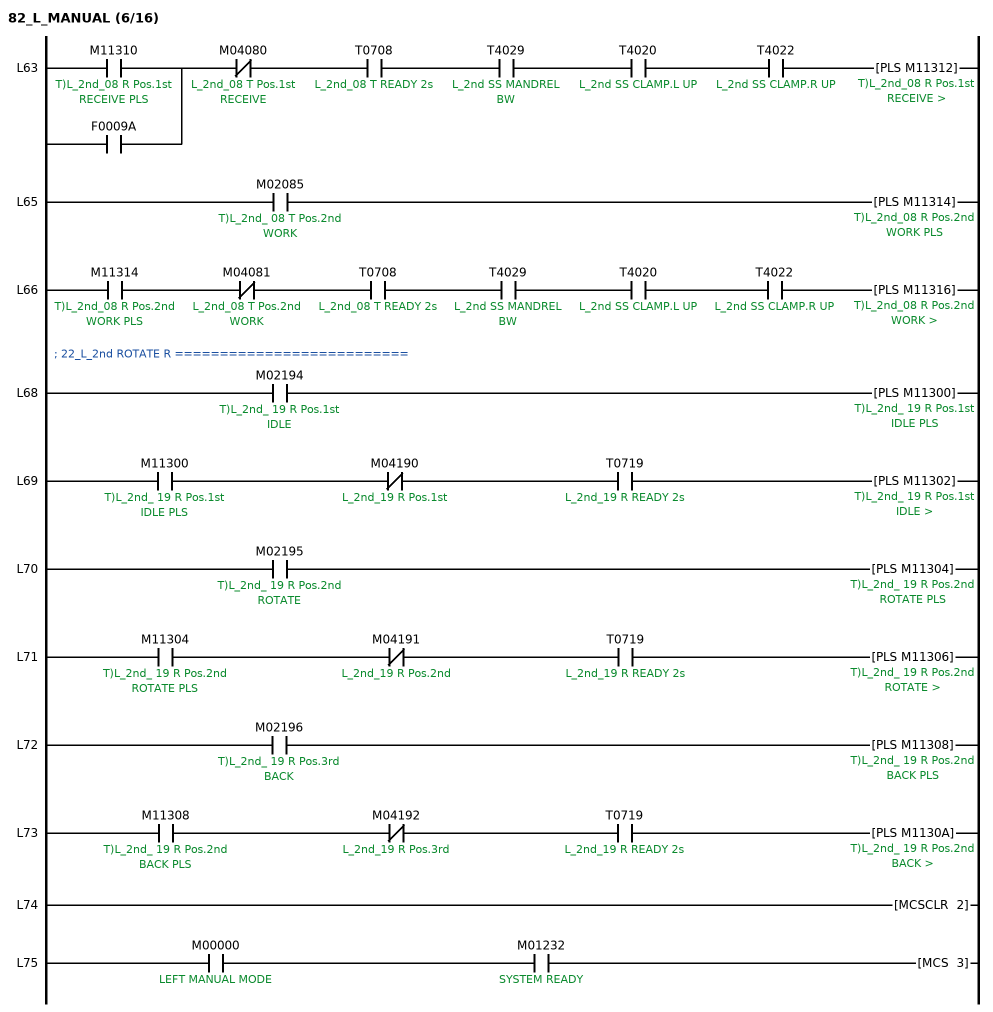
; L63
LOAD      M11310	// T)L_2nd_08 R Pos.1st RECEIVE PLS
OR        F0009A
AND NOT   M04080	// L_2nd_08 T Pos.1st RECEIVE
AND       T0708	// L_2nd_08 T READY 2s
AND       T4029	// L_2nd SS MANDREL BW
AND       T4020	// L_2nd SS CLAMP.L UP
AND       T4022	// L_2nd SS CLAMP.R UP
OUTP      M11312	// T)L_2nd_08 R Pos.1st RECEIVE >
; L65
LOAD      M02085	// T)L_2nd_ 08 T Pos.2nd WORK
OUTP      M11314	// T)L_2nd_08 R Pos.2nd WORK PLS
; L66
LOAD      M11314	// T)L_2nd_08 R Pos.2nd WORK PLS
AND NOT   M04081	// L_2nd_08 T Pos.2nd WORK
AND       T0708	// L_2nd_08 T READY 2s
AND       T4029	// L_2nd SS MANDREL BW
AND       T4020	// L_2nd SS CLAMP.L UP
AND       T4022	// L_2nd SS CLAMP.R UP
OUTP      M11316	// T)L_2nd_08 R Pos.2nd WORK >
// 22_L_2nd ROTATE R ==========================
; L68
LOAD      M02194	// T)L_2nd_ 19 R Pos.1st IDLE
OUTP      M11300	// T)L_2nd_ 19 R Pos.1st IDLE PLS
; L69
LOAD      M11300	// T)L_2nd_ 19 R Pos.1st IDLE PLS
AND NOT   M04190	// L_2nd_19 R Pos.1st 
AND       T0719	// L_2nd_19 R READY 2s
OUTP      M11302	// T)L_2nd_ 19 R Pos.1st IDLE >
; L70
LOAD      M02195	// T)L_2nd_ 19 R Pos.2nd ROTATE
OUTP      M11304	// T)L_2nd_ 19 R Pos.2nd ROTATE PLS
; L71
LOAD      M11304	// T)L_2nd_ 19 R Pos.2nd ROTATE PLS
AND NOT   M04191	// L_2nd_19 R Pos.2nd
AND       T0719	// L_2nd_19 R READY 2s
OUTP      M11306	// T)L_2nd_ 19 R Pos.2nd ROTATE >
; L72
LOAD      M02196	// T)L_2nd_ 19 R Pos.3rd BACK
OUTP      M11308	// T)L_2nd_ 19 R Pos.2nd BACK PLS
; L73
LOAD      M11308	// T)L_2nd_ 19 R Pos.2nd BACK PLS
AND NOT   M04192	// L_2nd_19 R Pos.3rd
AND       T0719	// L_2nd_19 R READY 2s
OUTP      M1130A	// T)L_2nd_ 19 R Pos.2nd BACK >
; L74
MCSCLR    2
; L75
LOAD      M00000	// LEFT MANUAL MODE
AND       M01232	// SYSTEM READY
MCS       3

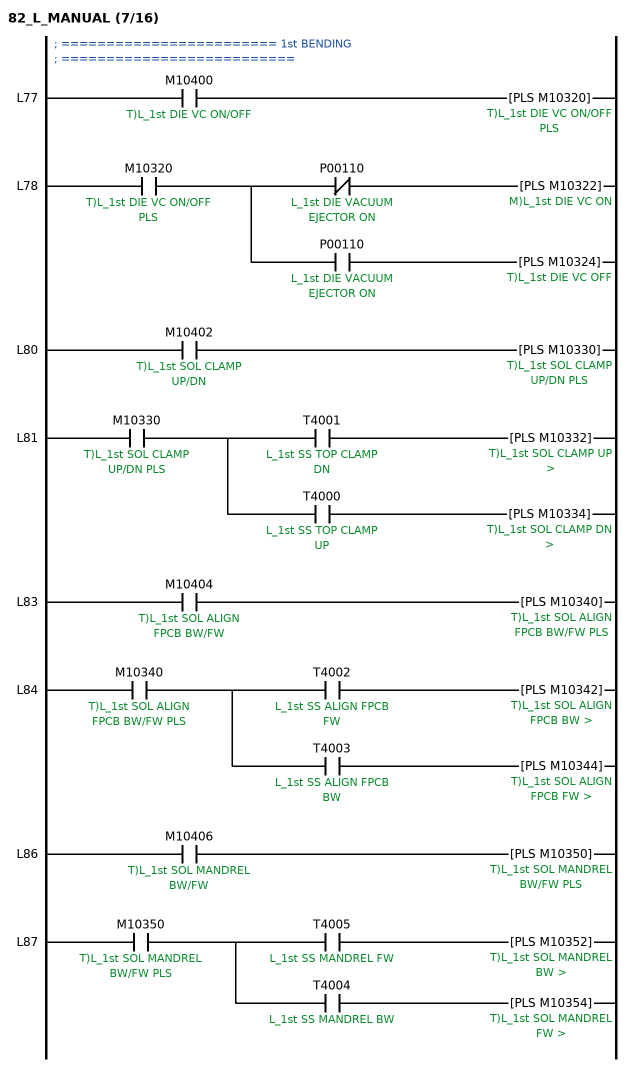
// ======================== 1st BENDING ==========================
; L77
LOAD      M10400	// T)L_1st DIE VC ON/OFF
OUTP      M10320	// T)L_1st DIE VC ON/OFF PLS
; L78
LOAD      M10320	// T)L_1st DIE VC ON/OFF PLS
MPUSH
AND NOT   P00110	// L_1st DIE VACUUM EJECTOR ON
OUTP      M10322	// M)L_1st DIE VC ON
MPOP
AND       P00110	// L_1st DIE VACUUM EJECTOR ON
OUTP      M10324	// T)L_1st DIE VC OFF
; L80
LOAD      M10402	// T)L_1st SOL CLAMP UP/DN
OUTP      M10330	// T)L_1st SOL CLAMP UP/DN PLS
; L81
LOAD      M10330	// T)L_1st SOL CLAMP UP/DN PLS
MPUSH
AND       T4001	// L_1st SS TOP CLAMP    DN
OUTP      M10332	// T)L_1st SOL CLAMP UP >
MPOP
AND       T4000	// L_1st SS TOP CLAMP    UP
OUTP      M10334	// T)L_1st SOL CLAMP DN >
; L83
LOAD      M10404	// T)L_1st SOL ALIGN FPCB BW/FW
OUTP      M10340	// T)L_1st SOL ALIGN FPCB BW/FW PLS
; L84
LOAD      M10340	// T)L_1st SOL ALIGN FPCB BW/FW PLS
MPUSH
AND       T4002	// L_1st SS ALIGN FPCB FW
OUTP      M10342	// T)L_1st SOL ALIGN FPCB BW >
MPOP
AND       T4003	// L_1st SS ALIGN FPCB BW
OUTP      M10344	// T)L_1st SOL ALIGN FPCB FW >
; L86
LOAD      M10406	// T)L_1st SOL MANDREL BW/FW
OUTP      M10350	// T)L_1st SOL MANDREL BW/FW PLS
; L87
LOAD      M10350	// T)L_1st SOL MANDREL BW/FW PLS
MPUSH
AND       T4005	// L_1st SS MANDREL FW
OUTP      M10352	// T)L_1st SOL MANDREL BW >
MPOP
AND       T4004	// L_1st SS MANDREL BW
OUTP      M10354	// T)L_1st SOL MANDREL FW >

